(* CODESYS project PPC-GD-14.project
   Title: PPC-GD
   Company: Hoeschl Automação e Controle Ltda

Project tree, tasks and I/O mapping:
  Dispositivo : 751-9402 WAGO Compact Controller 100, WAGO, order no. 751-9402, version 6.3.1.5
    application Application
      libraries: Standard, 3.5.18.0 (System); Util, 3.5.21.0 (System); WagoAppDatalogger, 1.0.5.6 (WAGO); SysTimeRtc, * (System); SysTime, 3.5.17.0 (System); SysTypes Interfaces, * (System); CAA Mathematics, * (CAA Technical Workgroup); WagoSolSolutionBuilder, 1.0.0.5 (WAGO); CmpBitmapPool, * (System); SysTimeCore, * (System); VisuDialogs, * (System)
      task VISU_TASK (cyclic, interval 200 ms, priority 15) calls VisuElems.Visu_Prg
      task MainTask (cyclic, interval 5 ms, priority 10, watchdog 100 ms x 5) calls MainProgram
      task AlarmManagerTask (cyclic, interval 50 ms, priority 15) calls AlarmManager.Alarm_Prg
      global variables PerVar
      Pages/
        visualisation Alarms
        visualisation Schedulle
        visualisation Supervision
        visualisation Template
        visualisation Comissioning
        visualisation Setup
      function block FB_WriteInv [ST]
      FB Auxiliares/
        function block FB_Scheduler [ST]
        function block FB_QAlloc [ST]
        function block FB_SafetyMargin [ST]
        function block FB_FFQ [ST]
        function block FB_DroopP [ST]
        function block FB_PI [ST]
        function block FB_FLimiter [ST]
        function block FB_PowerController [ST]
        function block FB_PIQ [ST]
        function block FB_PAlloc [ST]
        function block FB_Diagnostico [ST]
      image pool ImagePool
      function block FB_ReadMedidor [ST]
      program MainProgram [ST]
      function block FB_Controle [ST]
      function block FB_Startup [ST]
      global variables Global
      function block FB_ValidaDadosMedidor [ST]
      DataTypes/
        data type E_ModbusResult
        data type E_FailState
        data type UN_Real_to_Word_array
        data type ST_Rele
        data type UN_Medidor
        data type UN_Convert_Word_To_Real
        data type UN_Rele
        data type ST_Energia
        data type TTraceEntry
        data type E_StartupStatus
        data type E_MachineState
        data type UN_Energia
        data type ST_Medidor
        data type E_EventCode
      function block FB_Alarmes [ST]
      function block FB_ValidaDadosRele [ST]
      Alarm Configuration
        alarm class Warning (priority 50, acknowledge REP)
        alarm class Alarm (priority 30, acknowledge REP)
        AlarmStorage
        alarm class Critical (priority 0, acknowledge ACK)
        alarm group Startup
            0 []: Comparison Equal
        text list Startup
        alarm group Measurement
        text list Measurement
        alarm group InverterComms
        text list InverterComms
        alarm group Protection
        text list Protection
        alarm group StopTrip
        text list StopTrip
        alarm group SystemWatchdog
        text list SystemWatchdog
      global variables GVL_Alarm
    RS485_02 : Modbus COM, CODESYS, version 4.4.0.0
        settings: DataBits = 8; StopBits = 1; ComPort = 2
      Master_02 : Modbus Client, COM Port, CODESYS, version 4.5.0.0
          settings: Transmission = 'RTU'; ResponseTimeout = 150; TimeBetweenFrames = 10; Auto-restart communication = TRUE
        Inversor204 : Modbus Server, COM Port, CODESYS, version 4.5.0.0
            settings: SlaveAddress = 204; ResponseTimeout = 150; UseExtendedFunctionCodes = TRUE; Channel 0.Function Code = 16; Channel 0.Read Offset = 0; Channel 0.Read Length = 0; Channel 0.Write Offset = 16#0FA0; Channel 0.Write Length = 2; Channel 0.Cycle Time = 100
            output Application.Global.trigInvCOM200[4] : BIT  // Channel 0
            output Application.MainProgram.valor.Tw : ARRAY[0..1] OF WORD  // Channel 0
        Inversor203 : Modbus Server, COM Port, CODESYS, version 4.5.0.0
            settings: SlaveAddress = 203; ResponseTimeout = 150; UseExtendedFunctionCodes = TRUE; Channel 0.Function Code = 16; Channel 0.Read Offset = 0; Channel 0.Read Length = 0; Channel 0.Write Offset = 16#0FA0; Channel 0.Write Length = 2; Channel 0.Cycle Time = 100
            output Application.Global.trigInvCOM200[3] : BIT  // Channel 0
            output Application.MainProgram.valor.Tw : ARRAY[0..1] OF WORD  // Channel 0
        Inversor211 : Modbus Server, COM Port, CODESYS, version 4.5.0.0
            settings: SlaveAddress = 211; ResponseTimeout = 150; UseExtendedFunctionCodes = TRUE; Channel 0.Function Code = 16; Channel 0.Read Offset = 0; Channel 0.Read Length = 0; Channel 0.Write Offset = 16#0FA0; Channel 0.Write Length = 2; Channel 0.Cycle Time = 100
            output Application.Global.trigInvCOM200[11] : BIT  // Channel 0
            output Application.MainProgram.valor.Tw : ARRAY[0..1] OF WORD  // Channel 0
        Inversor201 : Modbus Server, COM Port, CODESYS, version 4.5.0.0
            settings: SlaveAddress = 201; ResponseTimeout = 150; UseExtendedFunctionCodes = TRUE; Channel 0.Function Code = 16; Channel 0.Read Offset = 0; Channel 0.Read Length = 0; Channel 0.Write Offset = 16#0FA0; Channel 0.Write Length = 2; Channel 0.Cycle Time = 100
            output Application.Global.trigInvCOM200[1] : BIT  // Channel 0
            output Application.MainProgram.valor.Tw : ARRAY[0..1] OF WORD  // Channel 0
        Inversor209 : Modbus Server, COM Port, CODESYS, version 4.5.0.0
            settings: SlaveAddress = 209; ResponseTimeout = 150; UseExtendedFunctionCodes = TRUE; Channel 0.Function Code = 16; Channel 0.Read Offset = 0; Channel 0.Read Length = 0; Channel 0.Write Offset = 16#0FA0; Channel 0.Write Length = 2; Channel 0.Cycle Time = 100
            output Application.Global.trigInvCOM200[9] : BIT  // Channel 0
            output Application.MainProgram.valor.Tw : ARRAY[0..1] OF WORD  // Channel 0
        Inversor212 : Modbus Server, COM Port, CODESYS, version 4.5.0.0
            settings: SlaveAddress = 212; ResponseTimeout = 150; UseExtendedFunctionCodes = TRUE; Channel 0.Function Code = 16; Channel 0.Read Offset = 0; Channel 0.Read Length = 0; Channel 0.Write Offset = 16#0FA0; Channel 0.Write Length = 2; Channel 0.Cycle Time = 100
            output Application.Global.trigInvCOM200[12] : BIT  // Channel 0
            output Application.MainProgram.valor.Tw : ARRAY[0..1] OF WORD  // Channel 0
        Inversor207 : Modbus Server, COM Port, CODESYS, version 4.5.0.0
            settings: SlaveAddress = 207; ResponseTimeout = 150; UseExtendedFunctionCodes = TRUE; Channel 0.Function Code = 16; Channel 0.Read Offset = 0; Channel 0.Read Length = 0; Channel 0.Write Offset = 16#0FA0; Channel 0.Write Length = 2; Channel 0.Cycle Time = 100
            output Application.Global.trigInvCOM200[7] : BIT  // Channel 0
            output Application.MainProgram.valor.Tw : ARRAY[0..1] OF WORD  // Channel 0
        Inversor213 : Modbus Server, COM Port, CODESYS, version 4.5.0.0
            settings: SlaveAddress = 213; ResponseTimeout = 150; UseExtendedFunctionCodes = TRUE; Channel 0.Function Code = 16; Channel 0.Read Offset = 0; Channel 0.Read Length = 0; Channel 0.Write Offset = 16#0FA0; Channel 0.Write Length = 2; Channel 0.Cycle Time = 100
            output Application.Global.trigInvCOM200[13] : BIT  // Channel 0
            output Application.MainProgram.valor.Tw : ARRAY[0..1] OF WORD  // Channel 0
        Medidor200 : Modbus Server, COM Port, CODESYS, version 4.5.0.0
            settings: SlaveAddress = 100; ResponseTimeout = 500; UseExtendedFunctionCodes = TRUE
        Inversor210 : Modbus Server, COM Port, CODESYS, version 4.5.0.0
            settings: SlaveAddress = 210; ResponseTimeout = 150; UseExtendedFunctionCodes = TRUE; Channel 0.Function Code = 16; Channel 0.Read Offset = 0; Channel 0.Read Length = 0; Channel 0.Write Offset = 16#0FA0; Channel 0.Write Length = 2; Channel 0.Cycle Time = 100
            output Application.Global.trigInvCOM200[10] : BIT  // Channel 0
            output Application.MainProgram.valor.Tw : ARRAY[0..1] OF WORD  // Channel 0
        Inversor208 : Modbus Server, COM Port, CODESYS, version 4.5.0.0
            settings: SlaveAddress = 208; ResponseTimeout = 150; UseExtendedFunctionCodes = TRUE; Channel 0.Function Code = 16; Channel 0.Read Offset = 0; Channel 0.Read Length = 0; Channel 0.Write Offset = 16#0FA0; Channel 0.Write Length = 2; Channel 0.Cycle Time = 100
            output Application.Global.trigInvCOM200[8] : BIT  // Channel 0
            output Application.MainProgram.valor.Tw : ARRAY[0..1] OF WORD  // Channel 0
        Inversor205 : Modbus Server, COM Port, CODESYS, version 4.5.0.0
            settings: SlaveAddress = 205; ResponseTimeout = 150; UseExtendedFunctionCodes = TRUE; Channel 0.Function Code = 16; Channel 0.Read Offset = 0; Channel 0.Read Length = 0; Channel 0.Write Offset = 16#0FA0; Channel 0.Write Length = 2; Channel 0.Cycle Time = 100
            output Application.Global.trigInvCOM200[5] : BIT  // Channel 0
            output Application.MainProgram.valor.Tw : ARRAY[0..1] OF WORD  // Channel 0
        Inversor215 : Modbus Server, COM Port, CODESYS, version 4.5.0.0
            settings: SlaveAddress = 215; ResponseTimeout = 150; UseExtendedFunctionCodes = TRUE; Channel 0.Function Code = 16; Channel 0.Read Offset = 0; Channel 0.Read Length = 0; Channel 0.Write Offset = 16#0FA0; Channel 0.Write Length = 2; Channel 0.Cycle Time = 100
            output Application.Global.trigInvCOM200[15] : BIT  // Channel 0
            output Application.MainProgram.valor.Tw : ARRAY[0..1] OF WORD  // Channel 0
        Inversor214 : Modbus Server, COM Port, CODESYS, version 4.5.0.0
            settings: SlaveAddress = 214; ResponseTimeout = 150; UseExtendedFunctionCodes = TRUE; Channel 0.Function Code = 16; Channel 0.Read Offset = 0; Channel 0.Read Length = 0; Channel 0.Write Offset = 16#0FA0; Channel 0.Write Length = 2; Channel 0.Cycle Time = 100
            output Application.Global.trigInvCOM200[14] : BIT  // Channel 0
            output Application.MainProgram.valor.Tw : ARRAY[0..1] OF WORD  // Channel 0
        Inversor202 : Modbus Server, COM Port, CODESYS, version 4.5.0.0
            settings: SlaveAddress = 202; ResponseTimeout = 150; UseExtendedFunctionCodes = TRUE; Channel 0.Function Code = 16; Channel 0.Read Offset = 0; Channel 0.Read Length = 0; Channel 0.Write Offset = 16#0FA0; Channel 0.Write Length = 2; Channel 0.Cycle Time = 100
            output Application.Global.trigInvCOM200[2] : BIT  // Channel 0
            output Application.MainProgram.valor.Tw : ARRAY[0..1] OF WORD  // Channel 0
        Inversor206 : Modbus Server, COM Port, CODESYS, version 4.5.0.0
            settings: SlaveAddress = 206; ResponseTimeout = 150; UseExtendedFunctionCodes = TRUE; Channel 0.Function Code = 16; Channel 0.Read Offset = 0; Channel 0.Read Length = 0; Channel 0.Write Offset = 16#0FA0; Channel 0.Write Length = 2; Channel 0.Cycle Time = 100
            output Application.Global.trigInvCOM200[6] : BIT  // Channel 0
            output Application.MainProgram.valor.Tw : ARRAY[0..1] OF WORD  // Channel 0
    Serial
      COM2 : COM2, WAGO, version 0.0.0.19 (disabled)
      COM1 : COM1, WAGO, version 0.0.0.19 (disabled)
    RS485_01 : Modbus COM, CODESYS, version 4.4.0.0
        settings: DataBits = 8; StopBits = 1; ComPort = 1
      Master_01 : Modbus Client, COM Port, CODESYS, version 4.5.0.0
          settings: Transmission = 'RTU'; ResponseTimeout = 150; TimeBetweenFrames = 10; Auto-restart communication = TRUE
        Inversor104 : Modbus Server, COM Port, CODESYS, version 4.5.0.0
            settings: SlaveAddress = 104; ResponseTimeout = 150; UseExtendedFunctionCodes = TRUE; Channel 0.Function Code = 16; Channel 0.Read Offset = 0; Channel 0.Read Length = 0; Channel 0.Write Offset = 16#0FA0; Channel 0.Write Length = 2; Channel 0.Cycle Time = 100
            output Application.Global.trigInvCOM100[4] : BIT  // Channel 0
            output Application.MainProgram.valor.Tw : ARRAY[0..1] OF WORD  // Channel 0
        Inversor105 : Modbus Server, COM Port, CODESYS, version 4.5.0.0
            settings: SlaveAddress = 105; ResponseTimeout = 150; UseExtendedFunctionCodes = TRUE; Channel 0.Function Code = 16; Channel 0.Read Offset = 0; Channel 0.Read Length = 0; Channel 0.Write Offset = 16#0FA0; Channel 0.Write Length = 2; Channel 0.Cycle Time = 100
            output Application.Global.trigInvCOM100[5] : BIT  // Channel 0
            output Application.MainProgram.valor.Tw : ARRAY[0..1] OF WORD  // Channel 0
        Inversor108 : Modbus Server, COM Port, CODESYS, version 4.5.0.0
            settings: SlaveAddress = 108; ResponseTimeout = 150; UseExtendedFunctionCodes = TRUE; Channel 0.Function Code = 16; Channel 0.Read Offset = 0; Channel 0.Read Length = 0; Channel 0.Write Offset = 16#0FA0; Channel 0.Write Length = 2; Channel 0.Cycle Time = 100
            output Application.Global.trigInvCOM100[8] : BIT  // Channel 0
            output Application.MainProgram.valor.Tw : ARRAY[0..1] OF WORD  // Channel 0
        Inversor101 : Modbus Server, COM Port, CODESYS, version 4.5.0.0
            settings: SlaveAddress = 101; ResponseTimeout = 150; UseExtendedFunctionCodes = TRUE; Channel 0.Function Code = 16; Channel 0.Read Offset = 0; Channel 0.Read Length = 0; Channel 0.Write Offset = 16#0FA0; Channel 0.Write Length = 2; Channel 0.Cycle Time = 100
            output Application.Global.trigInvCOM100[1] : BIT  // Channel 0
            output Application.MainProgram.valor.Tw : ARRAY[0..1] OF WORD  // Channel 0
        Inversor102 : Modbus Server, COM Port, CODESYS, version 4.5.0.0
            settings: SlaveAddress = 102; ResponseTimeout = 150; UseExtendedFunctionCodes = TRUE; Channel 0.Function Code = 16; Channel 0.Read Offset = 0; Channel 0.Read Length = 0; Channel 0.Write Offset = 16#0FA0; Channel 0.Write Length = 2; Channel 0.Cycle Time = 100
            output Application.Global.trigInvCOM100[2] : BIT  // Channel 0
            output Application.MainProgram.valor.Tw : ARRAY[0..1] OF WORD  // Channel 0
        Inversor112 : Modbus Server, COM Port, CODESYS, version 4.5.0.0
            settings: SlaveAddress = 112; ResponseTimeout = 150; UseExtendedFunctionCodes = TRUE; Channel 0.Function Code = 16; Channel 0.Read Offset = 0; Channel 0.Read Length = 0; Channel 0.Write Offset = 16#0FA0; Channel 0.Write Length = 2; Channel 0.Cycle Time = 100
            output Application.Global.trigInvCOM100[12] : BIT  // Channel 0
            output Application.MainProgram.valor.Tw : ARRAY[0..1] OF WORD  // Channel 0
        Inversor113 : Modbus Server, COM Port, CODESYS, version 4.5.0.0
            settings: SlaveAddress = 113; ResponseTimeout = 150; UseExtendedFunctionCodes = TRUE; Channel 0.Function Code = 16; Channel 0.Read Offset = 0; Channel 0.Read Length = 0; Channel 0.Write Offset = 16#0FA0; Channel 0.Write Length = 2; Channel 0.Cycle Time = 100
            output Application.Global.trigInvCOM100[13] : BIT  // Channel 0
            output Application.MainProgram.valor.Tw : ARRAY[0..1] OF WORD  // Channel 0
        Inversor110 : Modbus Server, COM Port, CODESYS, version 4.5.0.0
            settings: SlaveAddress = 110; ResponseTimeout = 150; UseExtendedFunctionCodes = TRUE; Channel 0.Function Code = 16; Channel 0.Read Offset = 0; Channel 0.Read Length = 0; Channel 0.Write Offset = 16#0FA0; Channel 0.Write Length = 2; Channel 0.Cycle Time = 100
            output Application.Global.trigInvCOM100[10] : BIT  // Channel 0
            output Application.MainProgram.valor.Tw : ARRAY[0..1] OF WORD  // Channel 0
        Medidor100 : Modbus Server, COM Port, CODESYS, version 4.5.0.0
            settings: SlaveAddress = 100; ResponseTimeout = 500; UseExtendedFunctionCodes = TRUE; Medidor.Function Code = 3; Medidor.Read Offset = 16#2006; Medidor.Read Length = 44; Medidor.Write Offset = 0; Medidor.Write Length = 0; Medidor.Cycle Time = 500
            output Application.Global.trigMedidor100 : BIT  // Medidor
            input  Application.MainProgram.fbReadMedidor.fbValidaDadosRele.valorLido.WordArray AT %IW7 : ARRAY[0..43] OF WORD  // Medidor
        Inversor103 : Modbus Server, COM Port, CODESYS, version 4.5.0.0
            settings: SlaveAddress = 103; ResponseTimeout = 150; UseExtendedFunctionCodes = TRUE; Channel 0.Function Code = 16; Channel 0.Read Offset = 0; Channel 0.Read Length = 0; Channel 0.Write Offset = 16#0FA0; Channel 0.Write Length = 2; Channel 0.Cycle Time = 100
            output Application.Global.trigInvCOM100[3] : BIT  // Channel 0
            output Application.MainProgram.valor.Tw : ARRAY[0..1] OF WORD  // Channel 0
        Inversor107 : Modbus Server, COM Port, CODESYS, version 4.5.0.0
            settings: SlaveAddress = 107; ResponseTimeout = 150; UseExtendedFunctionCodes = TRUE; Channel 0.Function Code = 16; Channel 0.Read Offset = 0; Channel 0.Read Length = 0; Channel 0.Write Offset = 16#0FA0; Channel 0.Write Length = 2; Channel 0.Cycle Time = 100
            output Application.Global.trigInvCOM100[7] : BIT  // Channel 0
            output Application.MainProgram.valor.Tw : ARRAY[0..1] OF WORD  // Channel 0
        Inversor115 : Modbus Server, COM Port, CODESYS, version 4.5.0.0
            settings: SlaveAddress = 115; ResponseTimeout = 150; UseExtendedFunctionCodes = TRUE; Channel 0.Function Code = 16; Channel 0.Read Offset = 0; Channel 0.Read Length = 0; Channel 0.Write Offset = 16#0FA0; Channel 0.Write Length = 2; Channel 0.Cycle Time = 100
            output Application.Global.trigInvCOM100[15] : BIT  // Channel 0
            output Application.MainProgram.valor.Tw : ARRAY[0..1] OF WORD  // Channel 0
        Inversor106 : Modbus Server, COM Port, CODESYS, version 4.5.0.0
            settings: SlaveAddress = 106; ResponseTimeout = 150; UseExtendedFunctionCodes = TRUE; Channel 0.Function Code = 16; Channel 0.Read Offset = 0; Channel 0.Read Length = 0; Channel 0.Write Offset = 16#0FA0; Channel 0.Write Length = 2; Channel 0.Cycle Time = 100
            output Application.Global.trigInvCOM100[6] : BIT  // Channel 0
            output Application.MainProgram.valor.Tw : ARRAY[0..1] OF WORD  // Channel 0
        Inversor114 : Modbus Server, COM Port, CODESYS, version 4.5.0.0
            settings: SlaveAddress = 114; ResponseTimeout = 150; UseExtendedFunctionCodes = TRUE; Channel 0.Function Code = 16; Channel 0.Read Offset = 0; Channel 0.Read Length = 0; Channel 0.Write Offset = 16#0FA0; Channel 0.Write Length = 2; Channel 0.Cycle Time = 100
            output Application.Global.trigInvCOM100[14] : BIT  // Channel 0
            output Application.MainProgram.valor.Tw : ARRAY[0..1] OF WORD  // Channel 0
        Inversor111 : Modbus Server, COM Port, CODESYS, version 4.5.0.0
            settings: SlaveAddress = 111; ResponseTimeout = 150; UseExtendedFunctionCodes = TRUE; Channel 0.Function Code = 16; Channel 0.Read Offset = 0; Channel 0.Read Length = 0; Channel 0.Write Offset = 16#0FA0; Channel 0.Write Length = 2; Channel 0.Cycle Time = 100
            output Application.Global.trigInvCOM100[11] : BIT  // Channel 0
            output Application.MainProgram.valor.Tw : ARRAY[0..1] OF WORD  // Channel 0
        Inversor109 : Modbus Server, COM Port, CODESYS, version 4.5.0.0
            settings: SlaveAddress = 109; ResponseTimeout = 150; UseExtendedFunctionCodes = TRUE; Channel 0.Function Code = 16; Channel 0.Read Offset = 0; Channel 0.Read Length = 0; Channel 0.Write Offset = 16#0FA0; Channel 0.Write Length = 2; Channel 0.Cycle Time = 100
            output Application.Global.trigInvCOM100[9] : BIT  // Channel 0
            output Application.MainProgram.valor.Tw : ARRAY[0..1] OF WORD  // Channel 0
    Compact Controller 100 Onboard IO
      X5_DIO : X5 DIO, WAGO, version 6.3.1.5
        X5_2 : SingleDO, WAGO, version 0.0.1.2
            output Application.Global.K2_out : BOOL  // _OUT
        X5_1 : SingleDO, WAGO, version 0.0.1.2
            output Application.Global.K1_out : BOOL  // _OUT
        X5_4 : SingleDO, WAGO, version 0.0.1.2
            output Application.Global.K4YellowOut : BOOL  // _OUT
        X5_7 : SingleDO, WAGO, version 0.0.1.2
            output Application.Global.K7OkOut : BOOL  // _OUT
        X5_8 : SingleDO, WAGO, version 0.0.1.2
            unmapped channels: _OUT
        X5_3 : SingleDO, WAGO, version 0.0.1.2
            output Application.Global.K3RedOut : BOOL  // _OUT
        X5_6 : SingleDO, WAGO, version 0.0.1.2
            unmapped channels: _OUT
        X5_5 : SingleDO, WAGO, version 0.0.1.2
            output Application.Global.K5GreenOut : BOOL  // _OUT
      X14_AIN : X14 AIN, WAGO, version 6.3.1.5
        X14_1 : SingleAI, WAGO, version 0.0.1.2
            unmapped channels: _PV
        X14_2 : SingleAI, WAGO, version 0.0.1.2
            unmapped channels: _PV
      X12_DI : X12 DI, WAGO, version 6.3.1.5
        X12_8 : Single DI, WAGO, version 0.0.1.2
            unmapped channels: _IN
        X12_3 : Single DI, WAGO, version 0.0.1.2
            unmapped channels: _IN
        X12_6 : Single DI, WAGO, version 0.0.1.2
            unmapped channels: _IN
        X12_4 : Single DI, WAGO, version 0.0.1.2
            unmapped channels: _IN
        X12_5 : Single DI, WAGO, version 0.0.1.2
            unmapped channels: _IN
        X12_2 : Single DI, WAGO, version 0.0.1.2
            input  Application.Global.K2_in : BOOL  // _IN
        X12_1 : Single DI, WAGO, version 0.0.1.2
            input  Application.Global.K1_in : BOOL  // _IN
        X12_7 : Single DI, WAGO, version 0.0.1.2
            unmapped channels: _IN
      X6_AIO : X6 AIO, WAGO, version 6.3.1.5
        X6_2 : SingleAI, WAGO, version 0.0.1.2
            unmapped channels: _PV
        X6_1 : SingleAI, WAGO, version 0.0.1.2
            unmapped channels: _PV
      X13_RTD : X13 RTD, WAGO, version 6.3.1.5
        X13_1 : SingleRTD, WAGO, version 0.0.1.2
            unmapped channels: _PV
        X13_2 : SingleRTD, WAGO, version 0.0.1.2
            unmapped channels: _PV
  libraries: VisuSymbols, 4.5.0.0 (System); WagoVisuIcons, 1.1.0.8 (WAGO); WagoVisuIconsMaterialDesign, 1.0.0.2 (WAGO)
  5ce3da45-db07-42e7-a21c-a00fff4ed8f6|Hacon logo + nome.jpeg
  text list GlobalTextList
  text list System
  5ce3da45-db07-42e7-a21c-a00fff4ed8f6|G:\Meu Drive\.02 Hacon-Solar\Marketing\Marca\HaconLogo.jpeg
*)

// Dispositivo/Application/DataTypes/E_ModbusResult
{attribute 'strict'}
TYPE E_ModbusResult :
(
    BUSY,   	// operação em andamento
    DONE,   	// leitura finalizada com sucesso (pulso curto)
    ERRO,   	// falha (permanece até reset)
	ABORT,		// comunicação foi abortada
	TIMEOUT,	// ocorreu TIMEOUT
	END			// finaliza a comunicação
);
END_TYPE

// Dispositivo/Application/DataTypes/E_FailState
{attribute 'qualified_only'}
{attribute 'strict'}
TYPE E_FailState :
(
    FS_INIT         := 0,  // Inicialização FAIL_SAFE
    FS_FORCE_ZERO   := 1,  // Forçar setpoint zero
    FS_WAIT_CONFIRM := 2,  // Aguardar confirmação escrita
    FS_VALIDATE     := 3,  // Validar geração zero
    FS_ESCALATE     := 4   // Escalar para STOP
) UINT;
END_TYPE

// Dispositivo/Application/DataTypes/UN_Real_to_Word_array
TYPE UN_Real_to_Word_array :
UNION
	RealArr  : ARRAY[1..15] OF REAL;   // 60 bytes
    WordArr  : ARRAY[1..30] OF WORD;   // 60 bytes
END_UNION
END_TYPE

// Dispositivo/Application/DataTypes/ST_Rele
TYPE ST_Rele :
	STRUCT
		//  22 variaveis do tipo real - ocupam 44 Words no array
		// variavel       tipo      modbusAddress origem         fator_escala 
		Ua    	    : REAL := 0.0; // 2006H - Tensão de fase A x 0,1 V
		Ub    	    : REAL := 0.0; // 2008H - Tensão de fase B x 0,1 V
		Uc    	    : REAL := 0.0; // 200AH - Tensão de fase C x 0,1 V
		Ia    	    : REAL := 0.0; // 200CH - Corrente de fase A x 0,001 A 
		Ib    	    : REAL := 0.0; // 200EH - Corrente de fase B x 0,001 A
		Ic    	    : REAL := 0.0; // 2010H - Corrente de fase C x 0,001 A
		Pt    	    : REAL := 0.0; // 2012H - Potencia ativa combinada x 0,1 W
		Pa    	    : REAL := 0.0; // 2014H - Potencia ativa fase A x 0,1 W
		Pb    	    : REAL := 0.0; // 2016H - Potencia ativa fase B x 0,1 W
		Pc    	    : REAL := 0.0; // 2018H - Potencia ativa fase C x 0,1 W	
		Qt    	    : REAL := 0.0; // 201AH - Potencia reativa combinada x 0,1 var
		Qa    	    : REAL := 0.0; // 201CH - Potencia reativa fase A x 0,1 var
		Qb    	    : REAL := 0.0; // 201EH - Potencia reativa fase B x 0,1 var
		Qc    	    : REAL := 0.0; // 2020H - Potencia reativa fase C x 0,1 var
		Reserved01  : REAL;        // 2022H - sem informação
		Reserved02  : REAL;        // 2024H - sem informação
		Reserved03  : REAL;        // 2026H - sem informação
		Reserved04  : REAL;        // 2028H - sem informação
		PFt    	    : REAL := 0.0; // 202AH - Fator de potência combinado (número positivo: indutivo, número negativo: capacitivo) (x  0,001)
		PFa    	    : REAL := 0.0; // 202CH - Fator de potência de fase A (número positivo: indutivo, número negativo: capacitivo)  (×0,001)
		PFb    	    : REAL := 0.0; // 202EH - Fator de potência de fase B (número positivo: indutivo, número negativo: capacitivo)  (×0,001)
		PFc    	    : REAL := 0.0; // 2030H - Fator de potência de fase C (número positivo: indutivo, número negativo: capacitivo)  (×0,001)
	END_STRUCT
END_TYPE

// Dispositivo/Application/DataTypes/UN_Medidor
TYPE UN_Medidor :
	UNION
        WordArray : ARRAY[0..43] OF WORD;
        EmReal    : ST_Rele;
    END_UNION
END_TYPE

// Dispositivo/Application/DataTypes/UN_Convert_Word_To_Real
TYPE UN_Convert_Word_To_Real :
	UNION
        Tw : ARRAY[0..1] OF WORD;
        Tr : REAL;
    END_UNION
END_TYPE

// Dispositivo/Application/DataTypes/UN_Rele
TYPE UN_Rele :
	UNION
        WordArray : ARRAY[0..43] OF WORD;
        EmReal    : ST_Rele;
    END_UNION
END_TYPE

// Dispositivo/Application/DataTypes/ST_Energia
TYPE ST_Energia :
	STRUCT
		// variavel       tipo      modbusAddress origem         fator_escala 
		EAImp  : REAL := 0.0; // 101EH - energia ativa total positiva (kWh)
		Vazia1 : REAL := 0.0; // 1020H - void
		Vazia2 : REAL := 0.0; // 1022H - void
		Vazia3 : REAL := 0.0; // 1024H - void
		Vazia4 : REAL := 0.0; // 1026H - void
		EAExp  : REAL := 0.0; // 1028H - energia ativa total negativa (kWh)	
	END_STRUCT
END_TYPE

// Dispositivo/Application/DataTypes/TTraceEntry
TYPE TTraceEntry :
STRUCT
        cyc         : UDINT;
        mode        : USINT;
        startEdge   : BOOL;
        xExecute    : BOOL;
        xAbort      : BOOL;
        xBusy       : BOOL;
        xDone       : BOOL;
        xError      : BOOL;
        xAborted    : BOOL;
        toQ         : BOOL;
        modbusErr   : UDINT;
        eResult     : E_ModbusResult;
    END_STRUCT
END_TYPE

// Dispositivo/Application/DataTypes/E_StartupStatus
{attribute 'qualified_only'}
{attribute 'strict'}
TYPE E_StartupStatus :
(
  stSeriais,		(* inicializa serias COM1 e COM2 *)
  stInit,			(* inicializa variaveis *)
  stWait_K1,      	(* transição imediata quando o delay completa *)
  stWait_K2,       	(* mantém bK3_out; monitora bK2_in com debounce *)
  stDone,           (* sucesso: desliga bK3_out e liga bK4_out *)
  stError           (* erro: sinaliza e coloca saídas em estado seguro *)
);
END_TYPE

// Dispositivo/Application/DataTypes/E_MachineState
{attribute 'qualified_only'}
{attribute 'strict'}
TYPE E_MachineState :
(
	START       := 0,  // inicializa o sistema uma única vez
    IDLE        := 1,  // Aguardando condições de início
    READ        := 2,  // Lendo medidor
    CONTROL     := 3,  // Calculando setpoints
    WRITE       := 4,  // Enviando comandos inversores
    FAIL	    := 5,  // Redução forçada (sem trip)
    STOP        := 6,   // Trip + latch (reset manual)
	ERROR       := 255 // Estado inválido/corrupto (fallback)
) UINT;
END_TYPE

// Dispositivo/Application/DataTypes/UN_Energia
TYPE UN_Energia :
	UNION
        WordArray : ARRAY[0..11] OF WORD;
        EmReal    : ST_Energia;
    END_UNION
END_TYPE

// Dispositivo/Application/DataTypes/ST_Medidor
TYPE ST_Medidor :
	STRUCT
		//  22 variaveis do tipo real - ocupam 44 Words no array
		// variavel       tipo      modbusAddress origem         fator_escala 
		Ua    	    : REAL := 0.0; // 2006H - Tensão de fase A x 0,1 V
		Ub    	    : REAL := 0.0; // 2008H - Tensão de fase B x 0,1 V
		Uc    	    : REAL := 0.0; // 200AH - Tensão de fase C x 0,1 V
		Ia    	    : REAL := 0.0; // 200CH - Corrente de fase A x 0,001 A 
		Ib    	    : REAL := 0.0; // 200EH - Corrente de fase B x 0,001 A
		Ic    	    : REAL := 0.0; // 2010H - Corrente de fase C x 0,001 A
		Pt    	    : REAL := 0.0; // 2012H - Potencia ativa combinada x 0,1 W
		Pa    	    : REAL := 0.0; // 2014H - Potencia ativa fase A x 0,1 W
		Pb    	    : REAL := 0.0; // 2016H - Potencia ativa fase B x 0,1 W
		Pc    	    : REAL := 0.0; // 2018H - Potencia ativa fase C x 0,1 W	
		Qt    	    : REAL := 0.0; // 201AH - Potencia reativa combinada x 0,1 var
		Qa    	    : REAL := 0.0; // 201CH - Potencia reativa fase A x 0,1 var
		Qb    	    : REAL := 0.0; // 201EH - Potencia reativa fase B x 0,1 var
		Qc    	    : REAL := 0.0; // 2020H - Potencia reativa fase C x 0,1 var
		Reserved01  : REAL;        // 2022H - sem informação
		Reserved02  : REAL;        // 2024H - sem informação
		Reserved03  : REAL;        // 2026H - sem informação
		Reserved04  : REAL;        // 2028H - sem informação
		PFt    	    : REAL := 0.0; // 202AH - Fator de potência combinado (número positivo: indutivo, número negativo: capacitivo) (x  0,001)
		PFa    	    : REAL := 0.0; // 202CH - Fator de potência de fase A (número positivo: indutivo, número negativo: capacitivo)  (×0,001)
		PFb    	    : REAL := 0.0; // 202EH - Fator de potência de fase B (número positivo: indutivo, número negativo: capacitivo)  (×0,001)
		PFc    	    : REAL := 0.0; // 2030H - Fator de potência de fase C (número positivo: indutivo, número negativo: capacitivo)  (×0,001)
	END_STRUCT
END_TYPE

// Dispositivo/Application/DataTypes/E_EventCode
{attribute 'qualified_only'}
{attribute 'strict'}
// ════════════════════════════════════════════════════════════════════
// E_EventCode — Código unificado de eventos do PPC-GD
// Compatível com Alarm Manager (flags BOOL em GVL_Alarm) e comissionamento.
// ════════════════════════════════════════════════════════════════════
//
// FAIXAS (nibble alto define severidade):
//   0x0000 = NONE
//   0X0xxx = ERROS    (Modbus driver)
//   0x1xxx = INFO     (registro operacional / transições)
//   0x2xxx = WARNING  (desvios toleráveis, sem ação de potência)
//   0x4xxx = ALARM    (falhas que requerem atenção / podem degradar)
//   0x8xxx = CRITICAL (ação de segurança: FAIL_SAFE ou STOP)
//
// 2º nibble = módulo:
//   x0xx = Sistema/Geral
//   x1xx = Startup
//   x2xx = Medição (medidor + validação)
//   x3xx = Comunicação inversores
//   x4xx = Controle (P/Q/PF)
//   x5xx = Scheduler/Agenda
//   x6xx = Máquina de Estados (MainProgram)
//   x7xx = Proteções normativas
//   x8xx = STOP/Trip
//   x9xx = Reservado
//
// Observação: códigos legados (ex-16#C1/C2/E1/E2/E3/F1) são referenciados
// por comentário e mapeados semanticamente, sem manter o mesmo valor numérico,
// para preservar a coerência de severidade por faixa.
// ════════════════════════════════════════════════════════════════════
TYPE E_EventCode :
(
    EVT_NONE                        := 16#0000,

    // =============================================================
    // INFO (0x1xxx)
    // =============================================================
    // ── Startup (0x11xx)
    INFO_STARTUP_BEGIN              := 16#1100,
    INFO_SERIAL_COM_OK              := 16#1101,
    INFO_RTC_OK                     := 16#1102,
    INFO_INVERTER_COUNT             := 16#1103,
    INFO_INSTALLED_POWER            := 16#1104,
    INFO_K1_CONFIRMED               := 16#1105,
    INFO_K2_CONFIRMED               := 16#1106,
    INFO_STARTUP_DONE               := 16#1107,

    // ── Medição / Operação (0x12xx)
    INFO_MEDIDOR_READ_OK            := 16#1200,
    INFO_MEDIDOR_DATA_VALID         := 16#1201,
    INFO_MEAS_RECOVERING            := 16#1202,  // contador nErrors reduzindo (opcional)

    // ── Escrita inversores (0x13xx)
    INFO_WRITE_INV_OK               := 16#1300,

    // ── Scheduler (0x15xx)
    INFO_SPECIAL_DATE_ACTIVE        := 16#1500,
    INFO_ZERO_GRID_MODE             := 16#1501,

    // ── Máquina de estados (0x16xx)
    INFO_STATE_CHANGE               := 16#1610,
    INFO_CYCLE_COMPLETE             := 16#1600,
    INFO_FAIL_RECOVERY              := 16#1601,

    // ── STOP/Reset (0x18xx)
    INFO_STOP_K2_OPEN_CONFIRMED     := 16#1800,
    INFO_STOP_RESET_APPROVED        := 16#1801,
    INFO_STOP_RESET_WAITING         := 16#1802,

    // =============================================================
    // WARNING (0x2xxx)
    // =============================================================
    // ── Startup
    WARN_TC_POWER_NOT_SET           := 16#2100,
    WARN_NO_INVERSORES_COM02        := 16#2101,

    // ── Medição
    WARN_MEAS_USING_LAST_VALID      := 16#2200,
    WARN_MEAS_ERROR_ISOLATED        := 16#2206,
    WARN_MEAS_CROSS_CHECK_PA        := 16#2201,
    WARN_MEAS_CROSS_CHECK_PB        := 16#2202,
    WARN_MEAS_CROSS_CHECK_PC        := 16#2203,
    WARN_MEAS_CROSS_CHECK_PT_SUM    := 16#2204,
    WARN_MEAS_CROSS_CHECK_PF        := 16#2205,

    // ── Comunicação inversores
    WARN_WRITE_INV_ERROR            := 16#2300,
    WARN_WRITE_INV_TIMEOUT          := 16#2301,

    // ── Controle
    WARN_P_ALLOC_SATURATED          := 16#2400,
    WARN_Q_LIMITED_BY_SMAX          := 16#2401,
    WARN_PF_BELOW_TARGET            := 16#2402,
    WARN_PF_NOT_ACHIEVABLE          := 16#2403,
    WARN_PI_P_SATURATED             := 16#2404,
    WARN_PI_Q_SATURATED             := 16#2405,
    WARN_PHASE_LIMITED              := 16#2406,

    // ── Ciclo / watchdog
    WARN_SCAN_OVERRUN               := 16#2600,

    // ── STOP/reset
    WARN_STOP_RESET_DENIED          := 16#2800,

    // =============================================================
    // ALARM (0x4xxx)
    // =============================================================
    // 0x00Bx — Aplicação Modbus (já existentes)
    ALARM_MB_ILLEGAL_FUNC         := 16#0001,
    ALARM_MB_ILLEGAL_ADDR         := 16#0002,
    ALARM_MB_ILLEGAL_VALUE        := 16#0003,
    ALARM_MB_SLAVE_FAILURE        := 16#0004,
    ALARM_MB_ACKNOWLEDGE          := 16#0005,
    ALARM_MB_SLAVE_BUSY           := 16#0006,
    ALARM_MB_MEMORY_PARITY        := 16#0008,
    ALARM_MB_GW_PATH_UNAVAIL      := 16#000A,
    ALARM_MB_GW_DEVICE_FAIL       := 16#000B,
    ALARM_MB_RESPONSE_TIMEOUT     := 16#00A1,
    ALARM_MB_RESPONSE_CRC         := 16#00A2,
    ALARM_MB_WRONG_SLAVE          := 16#00A3,
    ALARM_MB_WRONG_FC             := 16#00A4,
    ALARM_MB_TCP_ALARMOR          := 16#00A5,
    ALARM_MB_INVALID_DATA         := 16#00A6,
    ALARM_MB_INVALID_PROTOCOL     := 16#00A7,
    ALARM_MB_INVALID_HEADER       := 16#00A8,
    ALARM_MB_INVALID_PARAM        := 16#00A9,
    ALARM_MB_UNDEFINED            := 16#00FF,
    ALARM_MB_APP_ABORTED          := 16#00B1,
    ALARM_MB_APP_TIMEOUT          := 16#00B2,
    
    // ── Medição — Range/Freeze
    ALARM_MEAS_VOLTAGE_A_RANGE      := 16#4200,
    ALARM_MEAS_VOLTAGE_B_RANGE      := 16#4201,
    ALARM_MEAS_VOLTAGE_C_RANGE      := 16#4202,
    ALARM_MEAS_CURRENT_A_RANGE      := 16#4203,
    ALARM_MEAS_CURRENT_B_RANGE      := 16#4204,
    ALARM_MEAS_CURRENT_C_RANGE      := 16#4205,
    ALARM_MEAS_PT_RANGE             := 16#4206,
    ALARM_MEAS_PA_RANGE             := 16#4207,
    ALARM_MEAS_PB_RANGE             := 16#4208,
    ALARM_MEAS_PC_RANGE             := 16#4209,
    ALARM_MEAS_QT_RANGE             := 16#420A,
    ALARM_MEAS_QA_RANGE             := 16#420B,
    ALARM_MEAS_QB_RANGE             := 16#420C,
    ALARM_MEAS_QC_RANGE             := 16#420D,
    ALARM_MEAS_PFT_RANGE            := 16#420E,
    ALARM_MEAS_PFA_RANGE            := 16#420F,
    ALARM_MEAS_PFB_RANGE            := 16#4210,
    ALARM_MEAS_PFC_RANGE            := 16#4211,
    ALARM_MEAS_FROZEN               := 16#4212,

    // ── Comunicação medidor
    ALARM_MEDIDOR_MODBUS_ERROR      := 16#A220,
    ALARM_MEDIDOR_TIMEOUT           := 16#A221,

    // ── Comunicação inversores (canal degradado)
    ALARM_COM_CH1_DEGRADED          := 16#A300,
    ALARM_COM_CH2_DEGRADED          := 16#A301,

    // =============================================================
    // CRITICAL (0x8xxx)
    // =============================================================
    // ── Startup
    CRIT_SERIAL_INIT_FAILED         := 16#8100,
    CRIT_RTC_FAILED                 := 16#8101,
    CRIT_NO_INSTALLED_POWER         := 16#8102,
    CRIT_K1_TIMEOUT                 := 16#8103,

    // ── Medição
    CRIT_MEAS_PERSISTENT_FAIL       := 16#8200,  // ex-16#C1 (medição falha persistente)
    CRIT_MEDIDOR_COM_FAIL           := 16#8201,  // ex-16#C2 (erro/timeout Modbus medidor)

    // ── Comunicação inversores
    CRIT_COM_CHANNEL_FAIL           := 16#8300,  // ex-16#C2 (falha canal inversores >50%)

    // ── Controle
    CRIT_INSTALLED_POWER_ZERO       := 16#8400,

    // ── Scheduler
    CRIT_RTC_READ_FAIL              := 16#8500,
    CRIT_SCHEDULE_INDEX_INVALID     := 16#8501,

    // ── Watchdog
    CRIT_SCAN_WATCHDOG              := 16#8600,  // ex-16#F1

    // ── Proteções normativas
    CRIT_HARD_LIMIT_15S             := 16#8700,  // ex-16#E1
    CRIT_EXPORT_OVER_LPI_30S        := 16#8701,  // ex-16#E2
    CRIT_MEDIDOR_TIMEOUT_IN_FAIL    := 16#8702,  // ex-16#E3

    // ── STOP / Trip
    CRIT_STOP_ENTRY                 := 16#8800,
    CRIT_K2_DID_NOT_OPEN            := 16#8801,  // corrige bug (não reutiliza ex-E2)
    CRIT_STATE_CORRUPTION           := 16#8802

) UINT;
END_TYPE

// Dispositivo/Application/PerVar
{attribute 'qualified_only'}
VAR_GLOBAL PERSISTENT RETAIN

    // CONFIGURAÇÕES DO SISTEMA (Dados que não podem ser perdidos no desligamento)
    
    // --- Configuração dos Inversores ---
	NInversoresCOM01    : UINT :=0;
	NInversoresCOM02    : UINT :=0;
	
    // Potência nominal (kW) por tipo
    InvActivePower 		: ARRAY[1..Global.NMAXINVERSORES] OF REAL; 		// kW
    // Potência Aparente Máxima (kVA) por tipo 
    InvSmaxPower 		: ARRAY[1..Global.NMAXINVERSORES] OF REAL;		// kVA

    // --- Parâmetros de Controle de Exportação ---
    PowerMode 			: UINT := 2;      								// 0=Total, 1=Por Fase, 2=Ambos
	OperationMode		: BOOL := TRUE;									// FALSE=Export Control  TRUE=Zero Grid
	ControlMode			: UINT := 1;									// 0 = manual  1 = automatico (PI ativo)
    TotalMaxExport_kW 	: REAL := 0; 									// Limite físico total (kW)
    PhaseMaxExport_kW 	: REAL := 0; 									// Limite físico por fase (kW)

    (* 
	Regra prática para GD solar: Ti entre 5s e 20s. Mais rápido pode oscilar com a latência Modbus. 
	Mais lento perde capacidade de compensar nuvens passando.
	Ti é o Tempo Integral do controlador PI, também chamado de tempo de reset.
	Relação Ki= Kp / Ti   Então se você tem Kp = 1.0 e Ti = 10s => Ki=1.0/10 = 0.1 (por segundo)
	Na prática para seu sistema:
	Ti pequeno (ex: 2s) → integral age rápido → mais agressivo → risco de oscilação
	Ti grande (ex: 30s) → integral age devagar → mais conservador → lento para corrigir erro estacionário
	Ti = 10s → o controlador elimina o erro estacionário em aproximadamente 30 a 40 segundos (≈ 3-4 × Ti)
	Resumo em uma frase:
	Ti = 10s é "quanto tempo o integrador leva para alcançar a mesma força que o proporcional já deu instantaneamente".
	*)
	
	// --- Controle Droop (Potência Ativa) ---
	Droop_Enable     	: BOOL := TRUE;      							// Habilita droop
	K_Droop          	: REAL := 0.15;      							// kW/kW  (ex.: 0.05 = 5% de ganho)
	Deadband_Droop   	: REAL := 2.0;       							// % (erro menor não gera droop)
	Droop_Max        	: REAL := 0.4;       							// Fração da potência instalada (ex.: 0.6 = 60%)
	
	// --- Parâmetros do Controlador PI (Potência Ativa) ---
    Kp_P           		: REAL := 0.25;									// Recomendado: 0.1 a 1.0
																	    // Maior → resposta mais rápida, risco de oscilação
																	    // Menor → mais suave, mas mais lento
    Ki_P           		: REAL := 0.02;									// Recomendado: 0.02 a 0.1 - Com 1s de ciclo e tempo morto ~1,2–1,6s, integral muito alto oscila.
																		// Com T=1s: constante de tempo integral Ti = Kp/Ki = 12,5s
																	    // Significado: elimina erro estacionário em ~10 segundos
																	    // NUNCA > 0.2 com T=1s (oscilação garantida)
	RampUp_P 			: REAL := 15.0;           						// Rampa de subida (kW/s) - limitar a 15-20 kW/s por causa do sweep de setpoints nos inversores
	RampDown_P 			: REAL := 20.0;         						// Rampa de descida (kW/s) - RampDown_P ≤ 20–30 kW/s
    Deadband_P  		: REAL := 1.0;  								// % da potência instalada (ex: 1.0 = 1%)
	
    // --- Configuração de Fator de Potência (PF) e Reativos (Q) ---
    PF_target       	: REAL := 0.92; 								// Alvo |PF|
	PF_sign				: REAL := 1.0;
    // Parâmetros do PI de Correção de Q (Feedforward + Feedback)
    Kp_Q           		: REAL := 50.0;									// Recomendado: 20.0 a 100.0 kvar/pu_PF
																	    // Unidade: kvar por unidade de erro de PF
																	    // Ex: erro PF = 0.02 → P_term = 50 * 0.02 = 1.0 kvar
    Ki_Q           		: REAL := 5.0;									// Recomendado: 2.0 a 10.0 kvar/(pu_PF·s
																	    // Com T=1s: Ti = Kp/Ki = 10s => elimina erro em ~30-40s
																	    // Significado: corrige PF em ~10 segundos	
	RampUp_Q 			: REAL := 50.0;            						// Rampa de subida (kvar/s)
	RampDown_Q 			: REAL := 50.0;          						// Rampa de descida (kvar/s)
	Deadband_Q 			: REAL := 0.01;          						// Zona morta de PF (ex: 0.01 = ±0.01) — padrão para GD

    // --- Histerese de Habilitação ---
    HysteresisOn	   	: REAL := 0.01; 								// Liga controle acima de 1%
    HysteresisOff		: REAL := 0.01; 								// Desliga abaixo de 1%
		
    // --- Agenda Semanal (7 dias x 24 horas) e Datas Especiais
	bHorarioVerao 		: BOOL:= FALSE;									// se TRUE  = Horário de Verão Ativo (+1h)
    WeekSchedule_kW 	: ARRAY[1..7, 1..24] OF REAL; 					// (1=Dom 2=Seg 3=Ter 4=Quarta 5=Quinta 6=Sexta 7=Sábado) em kW
    DatasEspeciais   	: ARRAY[1..GLOBAL.NDATASESPECIAIS] OF DATE;		// inicializa com zeros
	SpecialDaySchedule 	: ARRAY[1..Global.NDATASESPECIAIS] OF REAL;		// cada data especial tem apenas um valor de potencia maxima valido para o dia inteiro

    // ════════════════════════════════════════════════════════════════
    // LIMITES FÍSICOS DO SISTEMA (Baseados no Transformador e Rede)
    // ════════════════════════════════════════════════════════════════
	// SafetyMargin_kW = SafetyMargin_pct × TC_Power_kW / 100 - Margem de segurança para compensar erro de TC perto de zero
	SafetyMargin_pct 	: REAL := 3.0;     								// Percentual do TC (%)
	// Exemplo 1: TC de 500 A, Tensão 380 V => P_TC = √3 × V × I = 1.732 × 380 × 500 = 329 kW
	TC_Power_kW			: REAL := 0.0; 									// deve ser configurado como 3% da potencia total sob controle pelo TC
	
	VMIN 				: REAL := 7170;  // Volts - tensão de fase minima para tensão primária de 13,8kV
    VMAX 				: REAL := 8370;  // Volts - tensão de fase máxima para tensão primária de 13,8kV
    IMAX 				: REAL := 125.0;  // Amperes - corrente de linha - para potencia de usina de 3MW erro transformador 5%
    PMAX 				: REAL := 3200.0; // kW (Demanda contratada + 10% de margem)
	QMAX				: REAL := 2400.0; // kvar tan(acos(0.8)) × Pmax
	// τ = tempo para atingir ~63% do valor final e T_scan = período de amostragem (1s no seu caso)
	// α = T_scan / (τ + T_scan)  => Alpha=0.5 => 3 segundos para atingir 95% do valor final
	// Item 2.1: "Responder em até 15 segundos a rejeição de carga"
	// Item 2.2: "Limitar exportação em até 15 segundos"
	// Nuvens passageiras: variação em 1–5 segundos
	// Rejeição de carga: instantânea (< 1s)
	// Ruído de medição: < 100 ms
	ALPHA				: REAL := 0.25;
	
END_VAR

// Dispositivo/Application/Global
{attribute 'qualified_only'}
VAR_GLOBAL CONSTANT

    // Parâmetros do sistema
    SOFTVERSION          		: UINT := 21;   				// Versão da aplicação
	DATAAPLICATION				: DATE := DATE#2025-12-05;		// Data da aplicação
	NMAXINVERSORES				: UINT := 30;					// Capacidade máxima de inversores
	TIPOSINVERSORES				: UINT := 8;					// total de inversores diferentes que podem estar presentes
	NDATASESPECIAIS 			: UINT := 48; 					// Quantidade de datas especiais disponíveis ao todo (para 10 anos)
	TIMEZONEOFFSET				: DINT := -3; 			
    CYCLE_TIME_MS				: UDINT := 1000;  				// tempo de ciclo de controle
	CYCLE_TIME_TOLERANCE		: UDINT := 1100;  				// tolerancia de ultrapassagem para tempo de ciclo de controle de 10%

END_VAR

VAR_GLOBAL
	timestampUTC				: UDINT;
	Result 						: RTS_IEC_RESULT;
	sMessage					: STRING(100) :='';
  	ControlCycle    			: REAL;            					// Tempo de ciclo de controle em SEGUNDOS (ex: 1.0 = 1 segundo)
	
	// Saidas digitais
  	K1_out  					: BOOL;   							// DI X5_1 - K1 - controle permissivo
	K2_out						: BOOL;								// DI X5_2 - K2 - controle trip
  	K3RedOut					: BOOL;								// DI X5_3 - nada pronto - acende vermelho
  	K4YellowOut  				: BOOL;   							// DI X5_4 - K2 aberto - acende amarelo
  	K5GreenOut  				: BOOL;   							// DI X5_5 - K2 fechou - acende verde
	K7OkOut  					: BOOL;   							// DI X5_7 - sinaliza ok
	K8ErroOut  					: BOOL;   							// DI X5_8 - sinaliza erro
		
	// Entredas digitais
	K1_in        				: BOOL;                				// DI X12_1 - contato auxliar de K1
  	K2_in        				: BOOL;                				// DI X12_2 - contato auxliar de K2

    //    Medições (REAL) - Tensões (V), Correntes (A), Potências Ativas (W), Potências Reativas (var), PF (adimensional, sinal: + indutivo, - capacitivo)
	
    Ua  			: REAL := 0.0; // Tensão de fase A   - 2006H - Tensão de fase A em Volts (x 0,1 V)
    Ub  			: REAL := 0.0; // Tensão de fase B   - 2008H - Tensão de fase B em Volts (x 0,1 V)
    Uc  			: REAL := 0.0; // Tensão de fase C   - 200AH - Tensão de fase C em Volts (x 0,1 V)
	
	Ia    			: REAL 	:= 0.0; // 200CH - Corrente de fase A em A (x 0,001 A) 
	Ib    			: REAL 	:= 0.0; // 200EH - Corrente de fase B em A (x 0,001 A) 
	Ic    			: REAL 	:= 0.0; // 2010H - Corrente de fase C em A (x 0,001 A) 
	
	Pt    			: REAL 	:= 0.0; // 2012H - Potencia ativa combinada em kW (x 0.1 para W, x 0.0001 para kW)
	Pa    			: REAL 	:= 0.0; // 2014H - Potencia ativa fase A 	em kW (x 0.1 para W, x 0.0001 para kW)
	Pb    			: REAL 	:= 0.0; // 2016H - Potencia ativa fase B 	em kW (x 0.1 para W, x 0.0001 para kW)
	Pc    			: REAL 	:= 0.0; // 2018H - Potencia ativa fase C    em kW (x 0.1 para W, x 0.0001 para kW)

	Qt    			: REAL 	:= 0.0; // 201AH - Potencia reativa combinada em kvar (x 0.1 para var, x 0.0001 para kvar)
	Qa    			: REAL 	:= 0.0; // 201CH - Potencia reativa fase A	 em kvar (x 0.1 para var, x 0.0001 para kvar)
	Qb    			: REAL 	:= 0.0; // 201EH - Potencia reativa fase B	 em kvar (x 0.1 para var, x 0.0001 para kvar)
	Qc    			: REAL 	:= 0.0; // 2020H - Potencia reativa fase C	 em kvar (x 0.1 para var, x 0.0001 para kvar)
	
	PFt    			: REAL 	:= 0.0; // 202AH - Fator de potência combinado (número positivo: indutivo, número negativo: capacitivo) (x0,001)
	PFa    			: REAL 	:= 0.0; // 202CH - Fator de potência de fase A (número positivo: indutivo, número negativo: capacitivo) (x0,001)
	PFb    			: REAL 	:= 0.0; // 202EH - Fator de potência de fase B (número positivo: indutivo, número negativo: capacitivo) (x0,001)
	PFc    			: REAL 	:= 0.0; // 2030H - Fator de potência de fase C (número positivo: indutivo, número negativo: capacitivo) (x0,001)	

    //   COMANDOS E TELEMETRIA - Saídas do Controle 
	
	// definição dos inversores dos dois canais de comunicação
	
	trigInvCOM100  	: ARRAY[1..15] OF BOOL;
    pInversores100 	: ARRAY [1..15] OF POINTER TO ModbusSlaveComPort; 				// array de pointers para Inversor01..Inversor15 (apenas ponteiros - não recria instâncias)
	trigMedidor100 	: BOOL;
	pMedidor100		: POINTER TO ModbusSlaveComPort;
	
	trigInvCOM200  	: ARRAY[1..15] OF BOOL;
	pInversores200 	: ARRAY [1..15] OF POINTER TO ModbusSlaveComPort; 				// array de pointers para Inversor01..Inversor15 (apenas ponteiros - não recria instâncias)
	trigMedidor200 	: BOOL;
	pMedidor200		: POINTER TO ModbusSlaveComPort;
	
	// Potencia Total instalada e potencia Aparente Total instalada
  	InstalledPower 	: REAL; 														// Soma da potência nominal de todos os inversores ativos
	Q_max_permitido : REAL := 0.0;    												// Q máximo permitido (kvar)
	InstalledSmax   : REAL; 														// NOVO: Potência Aparente Máxima Total (kVA)	
	
	// COMANDOS DE CONTROLE
	MaxExportLimit 	: REAL;              											// Limite de exportação do scheduler (kW)
	P_cmd_total_kW 	: REAL;              											// Comando total de P (kW)
	Q_cmd_total_kvar: REAL;            												// Comando total de Q (kvar)
	
    
    // Telemetria: Setpoint atual da agenda (antes das proteções)
    TotalPowerPercent : REAL;

    // Telemetria: Potência Reativa total desejada (kVA)
    TotalReactivePower : REAL;

    // Telemetria: Valores efetivos calculados para cada inversor
    P_inv_kW     	: ARRAY[1..NMAXINVERSORES] OF REAL; 							// valor de setpoint de potencia ativa em kW
	P_inv_Percent 	: ARRAY[1..NMAXINVERSORES] OF REAL; 							// valor de setpoint de potencia ativa em percentual do nominal
    Q_inv_kvar    	: ARRAY[1..NMAXINVERSORES] OF REAL; 							// valor de setpoint de potencia reativa em kVA
    PF_inv 			: ARRAY[1..NMAXINVERSORES] OF REAL; 							// valor do fator de potencia de cada inversor (deve ser 0,92 para todos)
	P_inv_limit 	: ARRAY[1..NMAXINVERSORES] OF REAL; 							// valor limite de potencia ativa com base na SMAX de cada um
	
	// Margem de segurança para compensar erro de TC perto de zero, o sistema tentará manter importação mínima garantido que não haja exportação
	SafetyMargin_pct: REAL :=0.03;
	TC_Power_kW		: REAL := 0.0; // deve ser configurado como 3% da potencia total sob controle pelo TC
	
	// ════════════════════════════════════════════════════════════════
	// DIAGNÓSTICO DE PF
	// ════════════════════════════════════════════════════════════════
	Q_available_max : REAL;             											// Q máximo disponível (kvar)
	PF_effective 	: REAL;                											// PF efetivo resultante
	PFErro 			: BOOL;                   										// TRUE = PF < 0.92 não atingível (banco de capacitores)
    
	// ════════════════════════════════════════════════════════════════
    // DIAGNÓSTICO DE FATOR DE POTÊNCIA
    // ════════════════════════════════════════════════════════════════
    
    // Status geral
    PF_target : REAL := 0.92;                   // PF alvo (mínimo aceitável)
    PF_measured : REAL;                         // PF medido no ponto de conexão
    PF_achieved : REAL;                         // PF efetivamente alcançado após compensação
    PF_OK : BOOL;                               // TRUE = PF ≥ 0.92
    
    // Potências
    P_generated_kW : REAL;                      // P total gerado pelos inversores
    P_allocated_kW : REAL;                      // P efetivamente alocado
    Q_measured_kvar : REAL;                     // Q medido no ponto de conexão (carga)
    Q_required_kvar : REAL;                     // Q necessário para atingir PF ≥ 0.92
    Q_commanded_kvar : REAL;                    // Q comandado pelo FB_PIQ
    Q_available_kvar : REAL;                    // Q que inversores conseguem fornecer
    Q_allocated_kvar : REAL;                    // Q efetivamente alocado
    Q_deficit_kvar : REAL;                      // Déficit de Q (se > 0, falta Q)
    
    // Capacidade dos inversores
    S_total_available_kVA : REAL;               // S total disponível (soma de todos inversores)
    S_total_used_kVA : REAL;                    // S total utilizado
    S_utilization_pct : REAL;                   // % de utilização de S
    Q_capacity_total_kvar : REAL;               // Capacidade total de Q dos inversores (atual)
    Q_utilization_pct : REAL;                   // % de utilização de Q
    
    // Diagnóstico e recomendações
    Q_deficit_percent : REAL;                   // Déficit de Q em % do necessário
    Capacitor_bank_size_kvar : REAL;            // Tamanho recomendado de banco de capacitores
    Capacitor_bank_recommended : BOOL;          // TRUE = Recomenda banco de capacitores
    PF_alarm_code : UINT;                       // Código de alarme (0=OK, 1=Aviso, 2=Crítico)
    PF_alarm_message : STRING(255);             // Mensagem descritiva do alarme
    
    // Histórico (opcional)
    PF_min_24h : REAL := 1.0;                   // PF mínimo nas últimas 24h
    PF_avg_24h : REAL := 1.0;                   // PF médio nas últimas 24h
    Q_deficit_max_24h : REAL;                   // Déficit máximo de Q nas últimas 24h
    PF_alarm_count_24h : UDINT;                 // Quantidade de alarmes nas últimas 24h
    
    // Inversores individuais (diagnóstico detalhado)
    Inv_S_utilization : ARRAY[1..NMAXINVERSORES] OF REAL;  // % S usado por inversor
    Inv_Q_available : ARRAY[1..NMAXINVERSORES] OF REAL;    // Q disponível por inversor (kvar)
    Inv_limited : ARRAY[1..NMAXINVERSORES] OF BOOL;        // TRUE = Inversor limitado por S	
END_VAR

// Dispositivo/Application/GVL_Alarm
{attribute 'qualified_only'}
VAR_GLOBAL
    // ─────────────────────────────────────────────────────────
    // ALARM MANAGER FLAGS (condições booleanas)
    // ─────────────────────────────────────────────────────────
    // Medição / Medidor
    ALM_MEAS_MEDIDOR_TIMEOUT       	: BOOL := FALSE;  // timeout de leitura (READ)
    ALM_MEDIDOR_MODBUS_ERRO        	: BOOL := FALSE;  // xError do medidor (READ)
    ALM_MEAS_PERSISTENT_FAIL		: BOOL := FALSE;  // bPoucosErros = FALSE
    ALM_MEAS_FROZEN	                : BOOL := FALSE;  // diagnosticCode = A900 (se aplicável)
    ALM_MEAS_USING_LAST_VALUEU		: BOOL := FALSE;  // bPoucosErros=TRUE e bDadosOK=FALSE
	ALM_MEAS_RANGE_ERROR    		: BOOL := FALSE;    // Warning: Valor fora de faixa
    ALM_MEAS_XCHECK_FAIL   			: BOOL := FALSE;    // Warning: Validação cruzada falhou

    // Comunicação inversores
    ALM_MODBUS_COM1_FAIL        	: BOOL := FALSE;  // >50% falhas COM1 no ciclo
    ALM_MODBUS_COM2_FAIL            : BOOL := FALSE;  // >50% falhas COM2 no ciclo
    ALM_COM_CHANNEL_FAIL           	: BOOL := FALSE;  // falha geral de comunicação → FAIL/STOP

    // Sistema
	ALM_SCAN_OVERRUN        		: BOOL := FALSE;    // Warning: Watchdog de ciclo
    ALM_RTC_FAIL            		: BOOL := FALSE;    // Error: Falha RTC
    ALM_NO_INVERTERS        		: BOOL := FALSE;    // Error: Nenhum inversor configurado
    ALM_INSTALLED_PWR_ZERO  		: BOOL := FALSE;    // Error: Potência instalada = 0
    ALM_TC_POWER_NOT_SET            : BOOL := FALSE;    // PerVar.TC_Power_kW = 0 na inicialização

    // Proteções normativas
    ALM_HARDLIMIT_15S       		: BOOL := FALSE;    // Error: P > LPI+10% por >15s
    ALM_EXPORT_30S          		: BOOL := FALSE;    // Error: P > LPI por >30s
    ALM_K2_NOT_OPENED       		: BOOL := FALSE;    // Error: K2 não abriu após trip
	
	// Status do sistema
    ALM_STOP_ACTIVE	                : BOOL := FALSE;  	// MachineState=STOP
	ALM_FAIL_ACTIVE					: BOOL := FALSE;  	// MachineState=FAIL

    // ── Controle / PF ──
    ALM_PF_BELOW_TARGET     		: BOOL := FALSE;    // Warning: PF < 0.92
    ALM_PF_CRITICAL         		: BOOL := FALSE;    // Error: PF < 0.92 + Q saturado
    ALM_Q_SATURATED         		: BOOL := FALSE;    // Info: Q limitado por S
END_VAR

// Dispositivo/Application/MainProgram
// DEBUG
// {#define DEBUG_MODE}
PROGRAM MainProgram
(*
    Máquina de estados principal do controlador.
    Fluxo geral:
    START   -> READ    (quando fbStart termina com sucesso)
    READ    -> CONTROL (quando leitura Modbus do medidor conclui OK)
    READ    -> IDLE    (quando leitura falha, mas ainda não estourou RETRIES_READ)
    READ    -> FAIL    (quando leitura falha e estoura RETRIES_READ)
    CONTROL -> WRITE   (sempre, um ciclo de controle por leitura)
    WRITE   -> IDLE    (depois de tentar escrever em todos inversores, se não estourou RETRIES_WRITE)
    WRITE   -> FAIL    (se falhas de escrita estourarem RETRIES_WRITE)
    IDLE    -> READ    (quando completar 1 segundo de ciclo)
    FAIL    -> (aguarda ação do operador)
    STOP    -> (parada controlada, permanece travado)
*)

VAR
    fbStart         		: FB_Startup;        		// executa a inicialização
    fbControle      		: FB_Controle;		 		// módulo de controle
	fbAlarmes				: FB_Alarmes;		 		// converte códigos de erros em mensagens texto
	fbChannel       		: ModbusChannel;
	fbReadMedidor 			: FB_ReadMedidor;
	fbWriteInvCOM1 			: FB_WriteInv;
    fbWriteInvCOM2 			: FB_WriteInv;
	
    // ══════════════════════════════════════════════════════════
    // Máquina de Estados
    // ══════════════════════════════════════════════════════════
	MachineState 			: E_MachineState := E_MachineState.START;
	MachineState_Last 		: E_MachineState := E_MachineState.START;
    FailState     			: E_FailState := E_FailState.FS_INIT;
	
    // ══════════════════════════════════════════════════════════
    // STOP: Trip e Reset Manual
    // ══════════════════════════════════════════════════════════
    StopLatch         : BOOL := FALSE;
    StopResetCmd      : BOOL := FALSE;
    StopEntryTime     : UDINT := 0;
    K2_CheckDone      : BOOL := FALSE;
    sMessage_K2       : STRING(100) := '';
    bResetConditionsOK: BOOL := FALSE;
    sResetDenialReason: STRING(255) := '';
    rTrigReset        : R_TRIG;
    tonResetWindow    : TON;

    // ══════════════════════════════════════════════════════════
    // Fault Codes
    // ══════════════════════════════════════════════==══════════
    FaultCode         : UINT := 0;
    FaultLatch        : BOOL := FALSE;
    
    // ══════════════════════════════════════════════════════════
    // Timers Normativos (DIS-NOR-033)
    // ══════════════════════════════════════════════════════════
    ton15s  : TON;   // Hard limit > 15s → STOP
    ton30s  : TON;   // Exportação > LPI por > 30s → STOP
    ton2s   : TON;   // Confirmação K2 aberto

    // ══════════════════════════════════════════════════════════
    // Health Monitoring
    // ══════════════════════════════════════════════════════════
    MedidorOK         : BOOL := FALSE;
    ComOK             : BOOL := FALSE;
    ComOK_COM1        : BOOL := TRUE;
    ComOK_COM2        : BOOL := TRUE;
    InvOnlineCount    : UINT := 0;
    ScanOverrunCount  : UINT := 0;
	
    // ══════════════════════════════════════════════════════════
    // Limites Calculados
    // ══════════════════════════════════════════════════════════
    LPI_per_phase_kW  : REAL := 0.0;
    HardLimit_mag     : REAL := 0.0;
    LPI_mag			  : REAL;
	Export_mag		  : REAL;
    // ══════════════════════════════════════════════════════════
    // Validação Cruzada
    // ══════════════════════════════════════════════════════════
    Pt_Last           : REAL := 0.0;
    P_inv_sum         : REAL := 0.0;
    
    // ══════════════════════════════════════════════════════════
    // Escrita em Inversores (Sequencial)
    // ══════════════════════════════════════════════════════════
    InvIndexCOM1      : UINT := 1;
    InvIndexCOM2      : UINT := 1;
    ErrorCountCOM1    : UINT := 0;
    ErrorCountCOM2    : UINT := 0;
    DoneCOM1          : BOOL := FALSE;
    DoneCOM2          : BOOL := FALSE;
    LastErrorIdxCOM1  : UINT := 0;
    LastErrorIdxCOM2  : UINT := 0;
    WriteErrorCOM1    : BOOL := FALSE;
    WriteErrorCOM2    : BOOL := FALSE;
    
    // ══════════════════════════════════════════════════════════
    // Temporização e Watchdog
    // ══════════════════════════════════════════════════════════
    tCycleStart       : UDINT := 0;
    tCycleEnd         : UDINT;
    tCycle            : UDINT;
    tElapsed          : UDINT;
    bFirstScanRead    : BOOL := TRUE;
    MaxCycleTime      : UDINT := 0;
    CycleTimeOverrunCount : UDINT := 0;
    
    // ══════════════════════════════════════════════════════════
    // Debug/Monitor
    // ══════════════════════════════════════════════════════════
    valor             : UN_Convert_Word_To_Real;
    auxvalor          : REAL := 0;
    stStart, stEnd, stCiclo : SYSTIME;
    tStartCom, tCom, tEndCom: SYSTIME;
    tMax              : SYSTIME := 0;
    Gatilho           : BOOL := TRUE;
    rTrigOn           : R_TRIG;
    fTrigOff          : F_TRIG;
    Primeiravez       : BOOL := TRUE;
    stCicloMax        : SYSTIME := 0;
    i                 : UINT;
    
    // ══════════════════════════════════════════════════════════
    // FAIL_SAFE (STOP Timeout)
    // ══════════════════════════════════════════════════════════
    tonStopWrite      : TON;
    tStopWrite        : TIME := T#2S;


	tonFailSafeRecovery		: TON;   // tempo para recuperação ao normal
	tonMedidorTimeout		: TON;   // tempo que aguarda medidor sem leitura
    
END_VAR


// ════════════════════════════════════════════════════════════════
// Atualiza Global.sMessage
// ════════════════════════════════════════════════════════════════
CASE MachineState OF
    E_MachineState.START: 	Global.sMessage := 'Inicializando';
	E_MachineState.IDLE: 	Global.sMessage := 'Aguardando';
    E_MachineState.READ:  	Global.sMessage := 'Operando - Leitura';
    E_MachineState.CONTROL: Global.sMessage := 'Operando - Control';
	E_MachineState.WRITE:	Global.sMessage := 'Operando - Setpoint';
    E_MachineState.STOP: 	Global.sMessage := 'STOP: Desconexão';	
    E_MachineState.FAIL:    Global.sMessage := 'Falha: Redução Forçada';
END_CASE

// ════════════════════════════════════════════════════════════════
// MÁQUINA DE ESTADOS PRINCIPAL
// ════════════════════════════════════════════════════════════════
CASE MachineState OF
	
// ────────────────────────────────────────────────────────────────
// START: Inicialização (fbStart + K1/K2)
E_MachineState.START:
    fbStart();  // Chamada do bloco de inicialização
	
	CASE fbStart.stState OF
  		E_StartupStatus.stSeriais,
		E_StartupStatus.stInit,
        E_StartupStatus.stWait_K1,
        E_StartupStatus.stWait_K2:
        	// Permanece em START
        E_StartupStatus.stDone:
			// Inicialização única (executada 1x após power-on)
			FailState := E_FailState.FS_INIT;
			FaultCode := 0;
			FaultLatch := FALSE;
			StopLatch := FALSE;
			ton15s(IN := FALSE);
			ton30s(IN := FALSE);
			ton2s(IN := FALSE);
            (* Inicialização concluída – segue para leitura *)		
            MachineState := E_MachineState.READ;

{#ifdef DEBUG_MODE}			
MachineState := E_MachineState.CONTROL;
auxvalor:=0;
{#endif}
	END_CASE;

// ────────────────────────────────────────────────────────────────
// READ: Leitura do Medidor
E_MachineState.READ:

    // Marca início do ciclo apenas uma vez ao entrar em READ
    IF bFirstScanRead THEN
        tCycleStart := SysTimeCore.SysTimeGetMs();
        bFirstScanRead := FALSE;
    END_IF;	
  	fbReadMedidor(Execute := TRUE);
	// avalia estado do Medidor a cada ciclo
	MedidorOK:=(fbReadMedidor.result = E_ModbusResult.DONE) AND fbReadMedidor.bDadosOK;
    IF fbReadMedidor.result = E_ModbusResult.DONE THEN
		IF MedidorOK THEN
            MachineState := E_MachineState.CONTROL;
        ELSE
            // ❌ Dados inválidos
            IF fbReadMedidor.bPoucosErros THEN
				// Erro isolado → continua com último valor válido
                MachineState := E_MachineState.CONTROL;
                Global.sMessage := 'MEDIÇÃO: Usando último válido';
			ELSE
                // Muitos erros → degradado
                MachineState := E_MachineState.FAIL;
                FaultCode := 16#C1;
                Global.sMessage := 'MEDIÇÃO: Falha persistente';
            END_IF
        END_IF
		
    ELSIF fbReadMedidor.result = E_ModbusResult.ERRO OR fbReadMedidor.result = E_ModbusResult.TIMEOUT THEN
		MachineState := E_MachineState.FAIL; 
        FaultCode := 16#C2;  
    END_IF

// ────────────────────────────────────────────────────────────────
// CONTROL: Cálculo de Setpoints
E_MachineState.CONTROL:
// Calcula setpoints (PI + droop)

IF Global.InstalledPower <= 0.0 THEN
	Global.sMessage := 'ERRO CRITICO: Potencia instalada = 0';
    Global.K8ErroOut := TRUE;
	MachineState := E_MachineState.STOP;
ELSE
	fbControle();  
END_IF

    // Inicialização da Escrita
    IF PerVar.NInversoresCOM01 > 0 THEN
        InvIndexCOM1 := 1;
        DoneCOM1 := FALSE;
    ELSE
        DoneCOM1 := TRUE;
		// SINALIZA ERRO
    END_IF;

    IF PerVar.NInversoresCOM02 > 0 THEN
        InvIndexCOM2 := 1;
        DoneCOM2 := FALSE;
    ELSE
        DoneCOM2 := TRUE;
    END_IF;

    MachineState := E_MachineState.WRITE;
{#ifdef DEBUG_MODE}	
MachineState := E_MachineState.CONTROL;
{#endif}

// ────────────────────────────────────────────────────────────────
// WRITE: Envia Comandos aos Inversores
E_MachineState.WRITE:
// Envia comandos aos inversores

{#ifdef DEBUG_MODE}	
	IF bFirstScanRead THEN
		tCycleStart := SysTimeCore.SysTimeGetMs();
		bFirstScanRead := FALSE;
	END_IF
{#endif}

	DoneCOM1 := (InvIndexCOM1 > PerVar.NInversoresCOM01);
	DoneCOM2 := (InvIndexCOM2 > PerVar.NInversoresCOM02);

    // COM1 (inversores 1..15)
    IF InvIndexCOM1 <= PerVar.NInversoresCOM01 THEN
        IF PerVar.InvActivePower[InvIndexCOM1] > 0.0 THEN
	{#ifdef DEBUG_MODE}
	// medição do tempo de execução
	rTrigOn(CLK := Global.pInversores100[1]^.xBusy);
	fTrigOff(CLK := Global.pInversores100[15]^.xBusy);
	(* Borda de subida → início *)
	IF rTrigOn.Q AND (InvIndexCOM1=1)   THEN
		SysTimeCore.SysTimeGetUs(tStartCom);
		Gatilho := TRUE;  // libera nova medição
	END_IF
	(* Borda de descida → fim *)
	IF fTrigOff.Q AND Gatilho THEN
		SysTimeCore.SysTimeGetUs(tEndCom);
		tCom := tEndCom - tStartCom; 
		IF tCom>tMax THEN
			tMax:=tCom;
		END_IF
		Gatilho := FALSE;
	END_IF
	{#endif}
            fbWriteInvCOM1(
                Execute := TRUE,
                InvIndex := InvIndexCOM1,
                trigInv := Global.trigInvCOM100[InvIndexCOM1],
                pSlave  := Global.pInversores100[InvIndexCOM1]^
            );

            IF (fbWriteInvCOM1.result = E_ModbusResult.DONE) THEN
                InvIndexCOM1 := InvIndexCOM1 + 1;
            ELSIF (fbWriteInvCOM1.result = E_ModbusResult.ERRO) OR
                  (fbWriteInvCOM1.result = E_ModbusResult.TIMEOUT) THEN
                // registra erro e continua
                ErrorCountCOM1 := ErrorCountCOM1 + 1;
                LastErrorIdxCOM1 := InvIndexCOM1;
                InvIndexCOM1 := InvIndexCOM1 + 1;
            END_IF
        ELSE
            // pular inversor inativo
            InvIndexCOM1 := InvIndexCOM1 + 1;
        END_IF
    ELSE
        DoneCOM1 := TRUE;
    END_IF

    // COM2 (inversores 16..30)
    IF InvIndexCOM2 <= PerVar.NInversoresCOM02 THEN
        IF PerVar.InvActivePower[InvIndexCOM2 + 15] > 0.0 THEN
            fbWriteInvCOM2(
                Execute := TRUE,
                InvIndex := InvIndexCOM2,
                trigInv := Global.trigInvCOM200[InvIndexCOM2],
                pSlave  := Global.pInversores200[InvIndexCOM2]^
            );

            IF (fbWriteInvCOM2.result = E_ModbusResult.DONE) THEN
                InvIndexCOM2 := InvIndexCOM2 + 1;
            ELSIF (fbWriteInvCOM2.result = E_ModbusResult.ERRO) OR
                  (fbWriteInvCOM2.result = E_ModbusResult.TIMEOUT) THEN
                // registra erro e continua
                ErrorCountCOM2 := ErrorCountCOM2 + 1;
                LastErrorIdxCOM2 := InvIndexCOM2;
                InvIndexCOM2 := InvIndexCOM2 + 1;
            END_IF
        ELSE
            // pular inversor inativo
            InvIndexCOM2 := InvIndexCOM2 + 1;
        END_IF
    ELSE
        DoneCOM2 := TRUE;
    END_IF

    // Fim da escrita
    IF DoneCOM1 AND DoneCOM2 THEN
        InvIndexCOM1 := 1;
        InvIndexCOM2 := 1;

        // ── Avaliar falhas por canal (>50% = falha do canal) ──
        IF PerVar.NInversoresCOM01 > 0 THEN
            ComOK_COM1 := (ErrorCountCOM1 <= (PerVar.NInversoresCOM01 / 2));
        ELSE
            ComOK_COM1 := TRUE;  // canal não utilizado = OK
        END_IF

        IF PerVar.NInversoresCOM02 > 0 THEN
            ComOK_COM2 := (ErrorCountCOM2 <= (PerVar.NInversoresCOM02 / 2));
        ELSE
            ComOK_COM2 := TRUE;  // canal não utilizado = OK
        END_IF

        // Qualquer canal ativo com falha → FAIL
        IF NOT ComOK_COM1 OR NOT ComOK_COM2 THEN
            FaultCode := 16#C2;
            MachineState := E_MachineState.FAIL;
        ELSE
            MachineState := E_MachineState.IDLE;
        END_IF
		// avalia o estado da comunicação com inversores
		ComOK:= (ComOK_COM1 AND ComOK_COM2);
        // Reset contadores para próximo ciclo
        ErrorCountCOM1 := 0;
        ErrorCountCOM2 := 0;
    END_IF

// ────────────────────────────────────────────────────────────────
// IDLE: Aguarda Completar Ciclo (1s)			
E_MachineState.IDLE:
//  Aguarda completar período de ciclo (1 segundo) depois de
	IF tCycleStart <> 0 THEN
    	tElapsed := SysTimeCore.SysTimeGetMs() - tCycleStart; 					// Calcula tempo desde início do ciclo
	END_IF;
	IF tElapsed >= GLOBAL.CYCLE_TIME_MS THEN
		MachineState := E_MachineState.READ;
		bFirstScanRead := TRUE;
       	// Atualiza estatísticas
       	IF tElapsed > MaxCycleTime THEN
           MaxCycleTime := tElapsed;
       	END_IF;  

	IF tElapsed > Global.CYCLE_TIME_TOLERANCE THEN
		ScanOverrunCount := ScanOverrunCount + 1;
		IF ScanOverrunCount >= 3 THEN
			FaultCode := 16#F1;  						// Watchdog scan
			MachineState := E_MachineState.FAIL;
			Global.sMessage := 'FAIL: Watchdog de ciclo';
			ScanOverrunCount := 0;
		END_IF
	ELSE
		ScanOverrunCount := 0;
	END_IF
{#ifdef DEBUG_MODE}
		MachineState := E_MachineState.CONTROL;
{#endif}
	END_IF;

// ────────────────────────────────────────────────────────────────
E_MachineState.FAIL:
// ESTADO FAIL — Redução forçada (norma DIS-NOR-033)
// ton15s: P > LPI + 10% Pnom por >15s → STOP
// ton30s: P > LPI por >30s → STOP

    // ══════════════════════════════════════════════════════════
    // TIMERS NORMATIVOS (monitorados TODO CICLO)
    // Cálculo do hard limit
	LPI_mag := ABS(Global.MaxExportLimit);
	Export_mag := MAX(0, -Global.Pt);
    HardLimit_mag := LPI_mag + (Global.InstalledPower * 0.1);
	
    // Mantém leitura do medidor (diagnóstico)
    fbReadMedidor(Execute := TRUE);
	
	// ✅ CORREÇÃO: Atualiza MedidorOK dentro de FAIL
    MedidorOK := (fbReadMedidor.result = E_ModbusResult.DONE) AND fbReadMedidor.bDadosOK;	
	
    // ── TIMER 15s: hard limit (P > LPI + 10% Pnom) ──
    ton15s(IN := (Export_mag > HardLimit_mag), PT := T#15S);

    // ── TIMER 30s: exportação persistente (P > LPI) ──
    ton30s(IN := (Export_mag > LPI_mag), PT := T#30S);
	
    // ── Escalada para STOP ──
    IF ton15s.Q OR ton30s.Q THEN
		IF ton15s.Q THEN
			FaultCode := 16#E1;  // hard limit: P > LPI + 10% Pnom por >15s
		ELSIF ton30s.Q THEN
			FaultCode := 16#E2;  // exportação > LPI por >30s
		END_IF
        MachineState := E_MachineState.STOP;
        RETURN;
    END_IF

    // ══════════════════════════════════════════════════════════
    // SUB-ESTADOS SIMPLIFICADOS
    CASE FailState OF

        E_FailState.FS_INIT:
		
			// Sinalização
			Global.K4YellowOut := TRUE;
			Global.K5GreenOut := FALSE;
            // Reinicializa índices de escrita
            InvIndexCOM1 := 1;
            InvIndexCOM2 := 1;
            DoneCOM1 := FALSE;
            DoneCOM2 := FALSE;
			ton15s(IN := FALSE);  
			ton30s(IN := FALSE);
			tonFailSafeRecovery(IN := FALSE);
			tonMedidorTimeout(IN := FALSE); 
            // Zera setpoints
            FOR i := 1 TO Global.NMAXINVERSORES DO
                Global.P_inv_kW[i] := 0.0;
                Global.P_inv_Percent[i] := 0.0;
                Global.Q_inv_kvar[i] := 0.0;
            END_FOR
            FailState := E_FailState.FS_FORCE_ZERO;
			Global.sMessage := 'Entrada em FAIL';

        E_FailState.FS_FORCE_ZERO:
            // Escreve zero em todos os inversores (mesmo código do WRITE, simplificado)
            DoneCOM1 := (InvIndexCOM1 > PerVar.NInversoresCOM01);
            DoneCOM2 := (InvIndexCOM2 > PerVar.NInversoresCOM02);

            // COM1
            IF NOT DoneCOM1 THEN
                IF PerVar.InvActivePower[InvIndexCOM1] > 0.0 THEN
                    fbWriteInvCOM1(
                        Execute := TRUE,
                        InvIndex := InvIndexCOM1,
                        trigInv := Global.trigInvCOM100[InvIndexCOM1],
                        pSlave  := Global.pInversores100[InvIndexCOM1]^
                    );
                    IF (fbWriteInvCOM1.result = E_ModbusResult.DONE) OR
                       (fbWriteInvCOM1.result = E_ModbusResult.ERRO) OR
                       (fbWriteInvCOM1.result = E_ModbusResult.TIMEOUT) THEN
                        InvIndexCOM1 := InvIndexCOM1 + 1;
                    END_IF
                ELSE
                    InvIndexCOM1 := InvIndexCOM1 + 1;
                END_IF
            END_IF

            // COM2
            IF NOT DoneCOM2 THEN
                IF PerVar.InvActivePower[InvIndexCOM2 + 15] > 0.0 THEN
                    fbWriteInvCOM2(
                        Execute := TRUE,
                        InvIndex := InvIndexCOM2,
                        trigInv := Global.trigInvCOM200[InvIndexCOM2],
                        pSlave  := Global.pInversores200[InvIndexCOM2]^
                    );
                    IF (fbWriteInvCOM2.result = E_ModbusResult.DONE) OR
                       (fbWriteInvCOM2.result = E_ModbusResult.ERRO) OR
                       (fbWriteInvCOM2.result = E_ModbusResult.TIMEOUT) THEN
                        InvIndexCOM2 := InvIndexCOM2 + 1;
                    END_IF
                ELSE
                    InvIndexCOM2 := InvIndexCOM2 + 1;
                END_IF
            END_IF

            // Escrita completa?
            IF DoneCOM1 AND DoneCOM2 THEN
                FailState := E_FailState.FS_VALIDATE;
            END_IF

        E_FailState.FS_VALIDATE:
            // Recuperação: P dentro da zona de controle (≤ LPI + 10% Pnom)
            IF (fbReadMedidor.result = E_ModbusResult.DONE) AND (Global.Pt >= -(Global.MaxExportLimit)) AND MedidorOK AND ComOK THEN
			   
				// ✅ Condições OK: conta tempo de recuperação
				tonFailSafeRecovery(IN := TRUE, PT := T#10S);
                IF tonFailSafeRecovery.Q THEN
                    // Recuperação automática
                    FailState := E_FailState.FS_INIT;
                    MachineState := E_MachineState.READ;
                    ton15s(IN := FALSE);
                    ton30s(IN := FALSE);
					tonMedidorTimeout(IN := FALSE);
            		tonFailSafeRecovery(IN := FALSE);
                    Global.K4YellowOut := FALSE;
                    Global.sMessage := 'Recuperação automática';
                END_IF				
            ELSE
        		// ❌ Condições NÃO OK: reseta recuperação e testa timeout
                tonFailSafeRecovery(IN := FALSE);
				// ❌ TIMEOUT de medidor (30s sem leitura válida)
                tonMedidorTimeout(IN := (fbReadMedidor.result <> E_ModbusResult.DONE), PT := T#30S);

                IF tonMedidorTimeout.Q THEN
					// ❌ STOP: Perda de visibilidade da planta
                    FaultCode := 16#E3;
                    MachineState := E_MachineState.STOP;
                    Global.sMessage := 'Timeout medidor em FAIL';
					tonMedidorTimeout(IN := FALSE);  // Reset timer
        			RETURN;
                END_IF
            END_IF
    END_CASE

// ────────────────────────────────────────────────────────────────
E_MachineState.STOP:
    // ══════════════════════════════════════════════════════════
    // A. ENTRADA EM STOP (primeira execução)
    // ══════════════════════════════════════════════════════════
    IF NOT StopLatch THEN
        StopLatch := TRUE;
        StopEntryTime := SysTimeCore.SysTimeGetMs();
        K2_CheckDone := FALSE;
        sMessage_K2 := '';
		        
        // Trip imediato
        Global.K2_out := TRUE;					// aciona trip do disjuntor
        Global.K1_out := FALSE;					// desliga bobina de minima tensão ou contator se existente
        Global.K3RedOut := TRUE;				// indica disjuntor desligado e houve falha
        Global.K4YellowOut := FALSE;
        Global.K5GreenOut := FALSE;
	    // zera setpoints por segurança
        FOR i := 1 TO Global.NMAXINVERSORES DO
            Global.P_inv_kW[i] := 0.0;
            Global.P_inv_Percent[i] := 0.0;
            Global.Q_inv_kvar[i] := 0.0;
        END_FOR	
	
    END_IF
    
    // ══════════════════════════════════════════════════════════
    // B. VERIFICAÇÃO DE K2 (executa apenas 1 vez)
    // ══==══════════════════════════════════════════════════════
    IF NOT K2_CheckDone THEN
        ton2s(IN := TRUE, PT := T#2S);
        
        IF ton2s.Q THEN
            K2_CheckDone := TRUE;
            ton2s(IN := FALSE);
            
            IF Global.K2_in = TRUE THEN
                Global.sMessage := CONCAT('STOP: ', 'CRITICO: K2 não abriu');
                FaultCode := 16#E2;
                FaultLatch := TRUE;
            ELSE
                Global.sMessage := CONCAT('STOP: ','K2 confirmado aberto');
                Global.K4YellowOut := TRUE;
            END_IF
        END_IF
    END_IF
    
    // ══════════════════════════════════════════════════════════
    // C. PROCESSAMENTO DE RESET MANUAL
    // ══════════════════════════════════════════════════════════
    rTrigReset(CLK := StopResetCmd);
    
	// Borda de subida: avalia condições básicas UMA VEZ
    IF rTrigReset.Q THEN
        // Avalia condições básicas
        bResetConditionsOK := (NOT Global.K2_in) AND (NOT FaultLatch) AND MedidorOK AND ComOK;      
		 IF NOT bResetConditionsOK THEN
			// Reset negado imediatamente
			StopResetCmd := FALSE;
			tonResetWindow(IN := FALSE);
			
			IF Global.K2_in THEN
				sResetDenialReason := 'K2 não está aberto';
			ELSIF FaultLatch THEN
				sResetDenialReason := 'FaultLatch ativo';
			ELSE
				sResetDenialReason := 'Medidor não OK';
			END_IF
			
			Global.sMessage := CONCAT('STOP reset NEGADO: ', sResetDenialReason);
		END_IF
	END_IF       
        
	// Monitoramento CONTÍNUO enquanto StopResetCmd=TRUE e condições OK
	IF StopResetCmd AND bResetConditionsOK THEN
		// Timer acumula enquanto Pt dentro do limite
		IF Global.MaxExportLimit > 0.0 THEN
			tonResetWindow(IN := (Global.Pt >= -(Global.MaxExportLimit)), PT := T#10S);
		ELSE
			tonResetWindow(IN := (Global.Pt > 0.0), PT := T#10S);
		END_IF
		
		IF tonResetWindow.Q THEN
			// ✅ Reset aprovado após 10s
			StopLatch := FALSE;
			StopResetCmd := FALSE;
			bResetConditionsOK := FALSE;
			MachineState := E_MachineState.START;
			FaultCode := 0;
			ton15s(IN := FALSE);
			ton30s(IN := FALSE);
			ton2s(IN := FALSE);
			tonResetWindow(IN := FALSE);
			Global.sMessage := 'STOP reset manual OK';
		ELSE
			Global.sMessage := 'Aguardando Pt estável por 10s...';
		END_IF	
	ELSE
		tonResetWindow(IN := FALSE);
	END_IF

END_CASE

END_PROGRAM

// Dispositivo/Application/FB_Startup
(* FB: fbStartup
   1) Ativa K1_out
   2) Aguarda 400 ms antes de verificar se K1_in está ativo
      -> Se K1_in NÃO estiver ativo depois deste tempo, sinaliza erro e sai da fbStartup
   3) Monitorar K2_in com debounce até ficar ativo 
   4) Enquanto aguarda K2_in ativar, mantém K4_out ativo
   5) Quando K2_in ativar (após debounced), desativa K4_out e ativa K5_out
   6) O controlador aguarda até K2_in = TRUE
   Notas:
   	- IMPORTANTE: se não forem usados contados auxiliares nos disjuntores, K1_in e K2_in precisam ser conectados a 24V
	- Este FB apenas sinaliza os outputs K1_out, K3_out, K4_out e K5_out.
   	- Implementado com máquina de estados e TONs (tDelay e tDebounce). TON deve ser chamado toda iteração.  *)
   
FUNCTION_BLOCK FB_Startup
VAR_OUTPUT
  stState			: E_StartupStatus:= E_StartupStatus.stSeriais;
END_VAR

VAR
  fbChannel       	: ModbusChannel;
  debouncedK1     	: BOOL := FALSE;   								// flag auxiliar informando que K1_in está estável em 1 
  TonDebounceK1     : TON;                          				// Novo timer debounce K1_in
  TimeDebounceK1    : TIME := T#500MS;              				// Tempo de debounce para K1

  debouncedK2 		: BOOL := FALSE; 								// flag auxiliar informando que K2_in está estável em 1 
  TonDebounceK2 	: TON;   										// timer para debounce de bk2 
  TimeDebounceK2    : TIME := T#500MS;     							// tempo de debounce para leitura de K2_in 
  
  cmdK01     		: BOOL := FALSE;  								// comandos calculados por ciclo e aplicados no final 
  auxRed     		: BOOL := FALSE;
  auxYellow     	: BOOL := FALSE;
  auxGreen     		: BOOL := FALSE;
  auxK1_in  		: BOOL;											// entradas digitais lidas no inicio da função 
  auxK2_in			: BOOL;
  indice			: UINT;
  
  // Variáveis para o Master 01 (COM1)
  eDeviceState01     		: DED.DEVICE_STATE; 					// Para guardar o estado retornado
  xDiagInfoIsAvailable01 	: BOOL;            						// Para guardar a saída xDiagnosisInfoAvailable
  eError01	      	    	: DED.ERROR;        					// Para guardar o código de erro
  xMaster01IsReady   		: BOOL;            						// Nosso booleano final de "pronto"
  
  // Variáveis para o Master 02 (COM2)
  eDeviceState02     		: DED.DEVICE_STATE; 					// Para guardar o estado retornado
  xDiagInfoIsAvailable02 	: BOOL;            						// Para guardar a saída xDiagnosisInfoAvailable
  eError02	           		: DED.ERROR;        					// Para guardar o código de erro
  xMaster02IsReady   		: BOOL;            						// Nosso booleano final de "pronto"
 

END_VAR

// INICIA AQUI

auxK1_in := Global.K1_in;
auxK2_in := Global.K2_in;

TonDebounceK1(IN := (stState = E_StartupStatus.stWait_K1) AND auxK1_in, PT := TimeDebounceK1); 	// debounce para K1_in
TonDebounceK2(IN := (stState = E_StartupStatus.stWait_K2) AND auxK2_in, PT := TimeDebounceK2);  // debounce para K2_in

CASE stState OF 																				// Máquina de estados

	E_StartupStatus.stSeriais:
		eDeviceState01 := Master_01.GetDeviceState(
			xDiagnosisInfoAvailable => xDiagInfoIsAvailable01,
			eError                  => eError01
			);
		eDeviceState02 := Master_02.GetDeviceState(
			xDiagnosisInfoAvailable => xDiagInfoIsAvailable02,
			eError                  => eError02
			);
  		xMaster01IsReady := (eDeviceState01 = DED.DEVICE_STATE.RUNNING); 
   		xMaster02IsReady := (eDeviceState02 = DED.DEVICE_STATE.RUNNING); 
		
		IF xMaster01IsReady AND xMaster02IsReady THEN
			stState := E_StartupStatus.stInit;
		ELSE
			stState := E_StartupStatus.stSeriais;
			// dispara Alarme por não conseguir abrir seriais
		END_IF
		
  	E_StartupStatus.stInit:																		// Inicialização única
	   
		cmdK01 			:= FALSE;
		auxRed  		:= FALSE;
		auxYellow 		:= FALSE;
		auxGreen  		:= FALSE;
		debouncedK1 	:= FALSE;
		debouncedK2 	:= FALSE;
		
		// Testa leitura do relógio do sistema na inicialização
		Global.timestampUTC := TO_UDINT(SysTimeRtcGet(Global.Result)); 							// UDINT#1528268918
		IF Global.Result <> eResultCode.OK THEN 												// Em caso de erro de leitura do relógio, zera a saída por segurança
			// sinalizar que houve erro para ler o relógio
			Global.K8ErroOut:=TRUE;
			RETURN;
		END_IF
	
		// Porta de comunicação COM1
		Global.pMedidor100   		:= ADR(Medidor100);
		Global.pInversores100[1]  	:= ADR(Inversor101);
		Global.pInversores100[2]  	:= ADR(Inversor102);
		Global.pInversores100[3]	:= ADR(Inversor103);
		Global.pInversores100[4] 	:= ADR(Inversor104);
		Global.pInversores100[5]	:= ADR(Inversor105);
		Global.pInversores100[6] 	:= ADR(Inversor106);
		Global.pInversores100[7] 	:= ADR(Inversor107);
		Global.pInversores100[8] 	:= ADR(Inversor108);
		Global.pInversores100[9] 	:= ADR(Inversor109);
		Global.pInversores100[10]	:= ADR(Inversor110);
		Global.pInversores100[11]	:= ADR(Inversor111);
		Global.pInversores100[12] 	:= ADR(Inversor112);
		Global.pInversores100[13] 	:= ADR(Inversor113);
		Global.pInversores100[14] 	:= ADR(Inversor114);
		Global.pInversores100[15] 	:= ADR(Inversor115);
		
		// Porta de comunicação COM2
		Global.pMedidor200   	  	:= ADR(Medidor200);
		Global.pInversores200[1]  	:= ADR(Inversor201);
		Global.pInversores200[2]  	:= ADR(Inversor202);
		Global.pInversores200[3]  	:= ADR(Inversor203);
		Global.pInversores200[4]  	:= ADR(Inversor204);
		Global.pInversores200[5] 	:= ADR(Inversor205);
		Global.pInversores200[6]  	:= ADR(Inversor206);
		Global.pInversores200[7]  	:= ADR(Inversor207);
		Global.pInversores200[8]  	:= ADR(Inversor208);
		Global.pInversores200[9]  	:= ADR(Inversor209);
		Global.pInversores200[10] 	:= ADR(Inversor210);
		Global.pInversores200[11] 	:= ADR(Inversor211);
		Global.pInversores200[12] 	:= ADR(Inversor212);
		Global.pInversores200[13] 	:= ADR(Inversor213);
		Global.pInversores200[14] 	:= ADR(Inversor214);
		Global.pInversores200[15] 	:= ADR(Inversor215);
		
		FOR indice := 1 TO 15 DO														// inicialização dos canais de comunicação
			fbChannel(Slave := Global.pInversores100[indice]^,xExecute := FALSE,xAbort := FALSE,iChannelIndex := 0);
			fbChannel(Slave := Global.pInversores200[indice]^,xExecute := FALSE,xAbort := FALSE,iChannelIndex := 0); 
		END_FOR
	
		// =========================================================================================
		// 0. PREPARAÇÃO DO TEMPO DE CICLO - feito na inicialização
		// =========================================================================================
		// Converte TIME (ex: T#500ms) para REAL (0.5 segundos) para uso nos PIDs
		Global.ControlCycle := UDINT_TO_REAL(Global.CYCLE_TIME_MS)/1000;  				// converte para segundos
			
		// ============================================================
		// CONTAGEM AUTOMÁTICA DE INVERSORES (sequencial por potência)
		// ============================================================
		
		// COM1: índices 1..15
		PerVar.NInversoresCOM01 := 0;
		FOR indice := 1 TO 15 DO
			IF PerVar.InvActivePower[indice] > 0.0 THEN
				PerVar.NInversoresCOM01 := indice;   // mantém maior índice válido
			ELSE
				EXIT;  // encontrou buraco -> encerra contagem
			END_IF
		END_FOR
		
		// COM2: índices 16..30
		PerVar.NInversoresCOM02 := 0;
		FOR indice := 16 TO 30 DO
			IF PerVar.InvActivePower[indice] > 0.0 THEN
				PerVar.NInversoresCOM02 := indice - 15;   // converte para faixa 1..15
			ELSE
				EXIT;  // encontrou buraco -> encerra contagem
			END_IF
		END_FOR		
		
		// =========================================================================================
		// 1. CÁLCULO DA POTÊNCIA INSTALADA TOTAL (Ativa e Aparente)  - feito na inicialização
		// =========================================================================================
		// Soma a capacidade nominal de todos os inversores configurados.
		// Isso permite mudar a planta dinamicamente sem recompilar.
		
		Global.InstalledPower := 0.0;
		Global.InstalledSmax  := 0.0;
		
		FOR indice := 1 TO Global.NMAXINVERSORES DO
			// Soma Potência Ativa Máxima (kW)
			Global.InstalledPower := Global.InstalledPower + PerVar.InvActivePower[indice];
			// Soma Potência Aparente Máxima (kVA)
			Global.InstalledSmax := Global.InstalledSmax + PerVar.InvSmaxPower[indice];
		END_FOR

		// Se não houver inversores ou potência válida, zera tudo e sai.
		IF Global.InstalledPower <= 0.0 THEN
			Global.TotalReactivePower := 0.0;
			// SINALIZA ALARME
			Global.K8ErroOut:=TRUE;
			RETURN;
		END_IF
		
		// Calcula Q_max_permitido 
	    Global.Q_max_permitido := Global.InstalledPower * 0.4256;  // tan(acos(0.92))
			
		// Configura TC_Power_kW se não foi configurado
		IF PerVar.TC_Power_kW = 0.0 THEN
			// SINALIZA ALARME
			Global.K8ErroOut:=TRUE;
			PerVar.TC_Power_kW := Global.InstalledPower;  // Aproximação conservadora
		END_IF

		// Muda para próximo estado	
		stState := E_StartupStatus.stWait_K1;

  E_StartupStatus.stWait_K1:															// DEBOUNCE K1
  
		cmdK01 := TRUE;
		auxRed := TRUE;																	// Status: aguardando K1 com debounce
		auxYellow := FALSE;
		auxGreen := FALSE;
		IF TonDebounceK1.Q THEN
		  debouncedK1 := TRUE;
		ELSE
		  debouncedK1 := FALSE;
		END_IF
	
		IF debouncedK1 THEN
		  stState := E_StartupStatus.stWait_K2;												// Somente avança se K1 está estabilizado
		  debouncedK2 := FALSE;
		  TonDebounceK1(IN := FALSE, PT := TimeDebounceK1); 								// (Opcional) reseta timer
		  auxRed := FALSE;																	// Status: aguardando K1 com debounce
		  auxYellow := TRUE;
		  auxGreen := FALSE;
		  
		END_IF

  E_StartupStatus.stWait_K2:	
  
		IF TonDebounceK2.Q THEN																// tDebounce.Q será TRUE se K2_in estável
		  debouncedK2 := TRUE;
		ELSE     																					
		  debouncedK2 := FALSE;																// se K2_in voltar a false, reseta timer
		END_IF
	
		IF debouncedK2 THEN
		  stState := E_StartupStatus.stDone;												// K2_ok e estável, processo de startup completo
		  TonDebounceK2(IN := FALSE, PT := TimeDebounceK2); 								// (Opcional) reseta timer
		  auxRed := FALSE;																	// Status: aguardando K1 com debounce
		  auxYellow := FALSE;
		  auxGreen := TRUE;
		END_IF
	
	E_StartupStatus.stDone:
	
		stState := E_StartupStatus.stDone;
		auxRed := FALSE;		
		auxYellow := FALSE;
		auxGreen := TRUE;

END_CASE;

//   Aplicar comandos calculados às saídas físicas / públicas
Global.K1_out 		:= cmdK01;
Global.K3RedOut 	:= auxRed;
Global.K4YellowOut 	:= auxYellow;
Global.K5GreenOut 	:= auxGreen;

END_FUNCTION_BLOCK

// Dispositivo/Application/FB_Controle
(*
   FB_Controle: Bloco Principal de Controle de Exportação (Zero Grid / Limitação).
   
   OBJETIVO:
   Gerenciar a potência ativa e reativa dos inversores para garantir que a exportação 
   de energia no ponto de conexão (PCC) não ultrapasse os limites definidos na agenda.

   ESTRATÉGIA DE CONTROLE (Lógica Inversa):
   - PV (Process Variable) é o valor medido no ponto de conexão
     - Valor Positivo (+) = Importando da rede (Consumo > Geração).
     - Valor Negativo (-) = Exportando para rede (Geração > Consumo).
   - SP (Set Point) é o limite de exportação (ex: -50kW).
   - O PID atua para manter PV >= SP.
     - Se PV > SP (Importando), o PID aumenta a geração.
     - Se PV < SP (Exportando), o PID reduz a geração.
	 Controle de Exportação em kW (Zero = Autoconsumo, Negativo = Exportação, Positivo = Importação).
	Erro: SP - PV.
	Ex: Quero exportar -10kW. Medidor lê +5kW (Importando). Erro = -10 - 5 = -15.
	Para aumentar a geração (reduzir a importação), o PID precisa agir. 
	Atenção: Como o comando do inversor é sempre positivo (0..100% de geração), a lógica interna do PI deve ser Inversa (Erro negativo -> Aumenta Saída) ou ajustamos o sinal do erro na entrada.
	
	No código abaixo, a estratégia usada foi de Normalizar o Erro para "Quanto falta gerar".
	Se o medidor diz +10kW (Importando), precisamos gerar +10kW a mais.
	Se o medidor diz -20kW (Exportando muito) e o limite é -10kW, precisamos gerar 10kW a menos.
	
    Hierarquia de prioridades ou objetivos:
	
    Prioridade 1: MAXIMIZAR P (Potência Ativa)
	Objetivo: Gerar o máximo de potência ativa possível
	Limite: Exportação máxima (agenda + safety margin + limite de fase)
	Flexibilidade: RÍGIDO - nunca exceder
	
	Prioridade 2: PF ≥ 0.92 NO PONTO DE CONEXÃO
	Objetivo: Manter fator de potência ≥ 0.92 (indutivo)
	Método: Compensar Q da carga com Q dos inversores
	Flexibilidade: SOFT - sinaliza se não conseguir, mas NÃO reduz P
	
	Prioridade 3: BALANCEAMENTO DE FASES
	
    
    Ordem de execução:
	0. Leitura do medidor e ajuste dos valores para unidades corretas 
	Lê registradores Modbus, converte e armazena como variáveis Globais
	
	Dentro de FB_Controle
	1. FB_Scheduler - Define limite de exportação baseado em datas, dias de semana e horário
    2. FB_PowertController
		2.1. PI → P_cmd_raw
    	2.2. Safety Margin → P_cmd_with_margin
    	2.3. Limitador de Fase → P_cmd_limited 
    3. FB_FFQ - Feedforward de Q (estimativa inicial)
    4. FB_PIQ - Controlador PI de fator de potência
	5. FB_PAlloc - Aloca P pelos inversores 
    6. FB_QAlloc - Aloca Q pelos inversores 
	7. FB_Diagnostico
	8. STATUS DE PF
*)
FUNCTION_BLOCK FB_Controle
VAR_INPUT
    bReset : BOOL;
END_VAR

VAR_OUTPUT
    bPF_OK : BOOL;
END_VAR

VAR
    // ════════════════════════════════════════════════════════════
    // SUBSISTEMAS (Function Blocks)
    // ════════════════════════════════════════════════════════════
    fbScheduler : FB_Scheduler;
    fbPowerCtrl : FB_PowerController;   // ✅ NOVO: Substitui fbPI + fbSafetyMargin + fbFLimiter
    fbFFQ : FB_FFQ;
    fbPIQ : FB_PIQ;
    fbPAlloc : FB_PAlloc;
    fbQAlloc : FB_QAlloc;
    fbDiagnostico : FB_Diagnostico;
    
    // ════════════════════════════════════════════════════════════
    // VARIÁVEIS DE TRABALHO
    // ════════════════════════════════════════════════════════════
    PF_measured : REAL;
    Q_cmd_kvar : REAL;
    Q_feedforward_kvar : REAL;
    bQ_limit_reached : BOOL := FALSE;
    bP_limit_reached : BOOL := FALSE;
END_VAR

// ════════════════════════════════════════════════════════════════
// 0. VERIFICAÇÕES INICIAIS E INICIALIZAÇÃO
// ════════════════════════════════════════════════════════════════
IF Global.InstalledPower <= 0.0 THEN
    // Sem potência instalada: zera todos os comandos
    bPF_OK := FALSE;
    Q_cmd_kvar := 0.0;
    Q_feedforward_kvar := 0.0;
    RETURN;  // Sai sem executar controle
END_IF

IF Global.InstalledSmax <= 0.0 THEN
    // Sem potência aparente: impossível calcular Q
    bPF_OK := FALSE;
    Q_cmd_kvar := 0.0;
    RETURN;
END_IF
// Fator de potência medido (valor absoluto)
PF_measured := ABS(Global.PFt);

// ════════════════════════════════════════════════════════════════
// 1. FB_SCHEDULER - Define Limite de Exportação
// ════════════════════════════════════════════════════════════════

IF PerVar.OperationMode THEN
	Global.MaxExportLimit:=0;				// TRUE = Zero Grid (exportação zero)
ELSE
	fbScheduler();   						// Global.MaxExportLimit definido a partir das agendas de horarios no Scheduller
END_IF

// ────────────────────────────────────────────────────────────────
// 2. CONTROLADOR DE POTÊNCIA ATIVA (PI + Safety + Limites)
// ────────────────────────────────────────────────────────────────

fbPowerCtrl(
    ExportLimit_kW := Global.MaxExportLimit,
    Feedback_kW := Global.Pt,
    bReset := bReset
);

bP_limit_reached := fbPowerCtrl.bPhase_limited OR fbPowerCtrl.bSaturated;
// ════════════════════════════════════════════════════════════════
// 3. FB_FFQ - Feedforward de Q 
// ════════════════════════════════════════════════════════════════

// Calcula Q necessário para manter PF = 0.92 com a potência comandada
fbFFQ(
    P_active_kW := fbPowerCtrl.P_cmd_kW, 
    PF_target_abs := PerVar.PF_target,
    PF_sign := 1.0                              // Indutivo (positivo)
);

Q_feedforward_kvar := fbFFQ.Q_reactive_kvar;  	

// ════════════════════════════════════════════════════════════════
// 4. FB_PIQ - Controle de Fator de Potência
// ════════════════════════════════════════════════════════════════

// Controlador PI de fator de potência
fbPIQ(
    SP := PerVar.PF_target,         							// Setpoint de PF (0.92)
    PV := PF_measured,              							// PF medido (absoluto)
	Kp:= PerVar.Kp_Q,
	Ki:= PerVar.Ki_Q,
	CycleTime:= Global.ControlCycle,
    P_cmd := fbPowerCtrl.P_cmd_kW,     							// Comando de P (para referência)
    RampUp := PerVar.RampUp_Q,      							// Rampa de subida (kvar/s)
    RampDown := PerVar.RampDown_Q,  							// Rampa de descida (kvar/s)
    DeadbandAbs := PerVar.Deadband_Q, 							// Zona morta de PF
    Reset := bReset,                 							// Reset
	bExternal_Saturated := bQ_limit_reached OR bP_limit_reached // FEEDBACK do ciclo anterior - calculado em fbQAlloc.
);

Q_cmd_kvar := Q_feedforward_kvar + fbPIQ.MV;  // Comando de Q em kvar

// Clamp superior: não pode exceder Q máximo dos inversores
IF Q_cmd_kvar > Global.Q_max_permitido THEN
    Q_cmd_kvar := Global.Q_max_permitido;
END_IF
// Clamp inferior: se PF_sign = indutivo, Q não pode ser negativo
IF Q_cmd_kvar < 0.0 THEN
    Q_cmd_kvar := 0.0;  // Não permite Q negativo (capacitivo) se não desejado
END_IF

// ════════════════════════════════════════════════════════════════
// 5. FB_PAlloc - Aloca P (PRIORIDADE MÁXIMA)
// ══════════���═════════════════════════════════════════════════════

fbPAlloc(
    P_total_cmd_kW := fbPowerCtrl.P_cmd_kW
);

Global.P_allocated_kW := fbPAlloc.P_allocated_kW;

// ════════════════════════════════════════════════════════════════
// 6. FB_QAlloc - Aloca Q 
// ════════════════════════════════════════════════════════════════

fbQAlloc(
    Q_total_cmd_kvar := Q_cmd_kvar
);

Global.Q_allocated_kvar := fbQAlloc.Q_allocated_kvar;

// Armazena flag de saturação para próximo ciclo
bQ_limit_reached := fbQAlloc.bQ_limit_reached;

// ════════════════════════════════════════════════════════════════
// 7. FB_Diagnostico - Gera diagnóstico completo
// ════════════════════════════════════════════════════════════════

fbDiagnostico(
    P_allocated_kW := fbPAlloc.P_allocated_kW,
    Q_commanded_kvar := Q_cmd_kvar,
    Q_allocated_kvar := fbQAlloc.Q_allocated_kvar,
    Q_capacity_kvar := fbQAlloc.Q_capacity_total,
    PF_measured := PF_measured,
    PF_achieved := fbQAlloc.PF_effective,
    bQ_limited := fbQAlloc.bQ_limit_reached
);

// ────────────────────────────────────────────────────────────────
// 8. STATUS DE PF
// ────────────────────────────────────────────────────────────────
IF fbQAlloc.PF_effective >= PerVar.PF_target THEN
    bPF_OK := TRUE;
ELSE
    bPF_OK := FALSE;
END_IF

END_FUNCTION_BLOCK

// Dispositivo/Application/FB Auxiliares/FB_Scheduler
(*
    FB_Scheduler
    - Agenda semanal: 24 intervalos por dia, 7 dias.
    - Recebe Hora UTC do sistema e converte internamente para LOCAL (Fuso + DST).
    - Feriados/datas especiais sobrescrevem a agenda.
    - Saída: setpoint % da potência instalada.
*)
FUNCTION_BLOCK FB_Scheduler

VAR
    // ════════════════════════════════════════════════════════════
    // VARIÁVEIS DE TIMESTAMP
    // ════════════════════════════════════════════════════════════
    timestampLocal_UDINT : UDINT;           // ✅ Apenas UDINT (sem DINT)
    offsetSeconds : DINT;                   // Offset em segundos (pode ser negativo)
    offsetSeconds_ABS : UDINT;              // Valor absoluto do offset
    
    // ════════════════════════════════════════════════════════════
    // CONVERSÕES DE DATA/HORA
    // ════════════════════════════════════════════════════════════
    dtNowLocal : DATE_AND_TIME;
    dataNowLocal : DATE;
    todNowLocal : TOD;
    todAsDword : DWORD;
    hora : INT;
    diadasemana : INT;
    
    // ════════════════════════════════════════════════════════════
    // CACHE DE DATAS ESPECIAIS (Otimização)
    // ════════════════════════════════════════════════════════════
    lastCheckedDate : DATE := DATE#1970-01-01;      // Última data verificada
    cachedSpecialDateLimit : REAL := -1.0;          // -1 = inválido
    
    // ════════════════════════════════════════════════════════════
    // AUXILIARES
    // ════════════════════════════════════════════════════════════
    i : UINT;
END_VAR


// ════════════════════════════════════════════════════════════════
// 1. LEITURA DO RELÓGIO DO SISTEMA (UTC)
// ════════════════════════════════════════════════════════════════

Global.timestampUTC := TO_UDINT(SysTimeRtcGet(Global.Result));

IF Global.Result <> eResultCode.OK THEN
    // ❌ ERRO: Relógio não disponível
    Global.MaxExportLimit := 0.0;
    Global.sMessage := 'ERRO CRITICO: Falha ao ler RTC';
    Global.K8ErroOut := TRUE;
    RETURN;
END_IF

// ════════════════════════════════════════════════════════════════
// 2. CÁLCULO DO OFFSET TOTAL (Fuso + Horário de Verão)
// ════════════════════════════════════════════════════════════════

// Offset base (fuso horário em segundos)
offsetSeconds := Global.TIMEZONEOFFSET * 3600;  // Ex: -3 * 3600 = -10800

// Adiciona horário de verão se ativo
IF PerVar.bHorarioVerao THEN
    offsetSeconds := offsetSeconds + 3600;      // +1 hora
END_IF

